KUKA KRL program: MyProgram_271().src

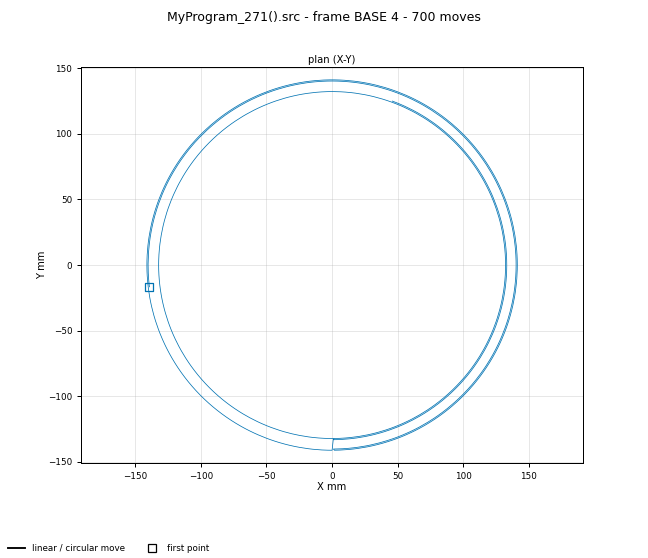
[picture p0: tool path of MyProgram_271().src in frame BASE 4, 700 of 700 moves have a stored position in this frame; points joined in program order, loops and branches not executed]
&ACCESS RVP
&REL 1
&PARAM TEMPLATE = C:\KRC\Roboter\Template\vorgabe
&PARAM EDITMASK = *
DEF MyProgram_271()
; ---- Setting reference (Base) ----
$BASE = BASE_DATA[4]

; --------------------------
; ---- Setting tool (TCP) ----
$TOOL = TOOL_DATA[3]
; --------------------------

$VEL.CP = VEL_APROX_PRINT
Startdeposition()
$VEL.CP = VEL_PRINT
LIN {X -139.2462,Y -16.5894,Z 170,A -172.5536,B 9.2163,C 0.2811,E1 9.0612,E2 264.1898} C_DIS
LIN {X -139.7898,Y -11.1357,Z 170,A -174.0658,B 9.2169,C 0.2622,E1 9.0608,E2 265.6084} C_DIS
LIN {X -140.1038,Y -5.997,Z 170,A -176.402,B 9.2169,C 0.2602,E1 9.0605,E2 267.9721} C_DIS
LIN {X -140.2304,Y 0.6703,Z 170,A -179.1601,B 9.2171,C 0.2528,E1 9.0604,E2 270.732} C_DIS
LIN {X -139.8512,Y 10.3146,Z 170,A 176.042,B 9.2171,C 0.2559,E1 9.0611,E2 275.6332} C_DIS
LIN {X -139.2175,Y 16.8301,Z 170,A 174.2066,B 9.2176,C 0.2339,E1 9.0617,E2 277.3608} C_DIS
LIN {X -138.6579,Y 20.951,Z 170,A 172.3266,B 9.2176,C 0.2321,E1 9.0624,E2 279.2619} C_DIS
LIN {X -137.8969,Y 25.4847,Z 170,A 170.0862,B 9.2176,C 0.2329,E1 9.0635,E2 281.5459} C_DIS
LIN {X -137.0475,Y 29.71,Z 170,A 168.7917,B 9.218,C 0.2199,E1 9.0643,E2 282.78} C_DIS
LIN {X -136.272,Y 33.0857,Z 170,A 167.3335,B 9.218,C 0.2166,E1 9.0652,E2 284.2422} C_DIS
LIN {X -135.2865,Y 36.9171,Z 170,A 165.7161,B 9.2181,C 0.2121,E1 9.0663,E2 285.8581} C_DIS
LIN {X -134.3405,Y 40.224,Z 170,A 164.2872,B 9.2182,C 0.2085,E1 9.0675,E2 287.2885} C_DIS
LIN {X -133.4935,Y 42.9443,Z 170,A 163.0667,B 9.2182,C 0.2062,E1 9.0685,E2 288.5149} C_DIS
LIN {X -132.1554,Y 46.9048,Z 170,A 161.2655,B 9.2183,C 0.2031,E1 9.0702,E2 290.3261} C_DIS
LIN {X -130.6875,Y 50.8469,Z 170,A 159.6638,B 9.2185,C 0.1964,E1 9.0717,E2 291.9111} C_DIS
LIN {X -129.48,Y 53.8478,Z 170,A 158.2691,B 9.2185,C 0.1941,E1 9.0732,E2 293.3137} C_DIS
LIN {X -128.0071,Y 57.2608,Z 170,A 156.6772,B 9.2185,C 0.1913,E1 9.075,E2 294.9132} C_DIS
LIN {X -126.4175,Y 60.6901,Z 170,A 155.1673,B 9.2187,C 0.1866,E1 9.0768,E2 296.4171} C_DIS
LIN {X -124.9093,Y 63.736,Z 170,A 153.7709,B 9.2187,C 0.1831,E1 9.0785,E2 297.813} C_DIS
LIN {X -123.2104,Y 66.9657,Z 170,A 152.1863,B 9.2187,C 0.1809,E1 9.0806,E2 299.4079} C_DIS
LIN {X -120.9477,Y 70.9706,Z 170,A 149.4715,B 9.2187,C 0.1905,E1 9.0846,E2 302.2246} C_DIS
LIN {X -117.5668,Y 76.4409,Z 170,A 147.5825,B 9.219,C 0.1713,E1 9.0873,E2 304.0192} C_DIS
LIN {X -114.9933,Y 80.2604,Z 170,A 145.6572,B 9.219,C 0.1675,E1 9.0904,E2 305.948} C_DIS
LIN {X -112.3015,Y 83.9859,Z 170,A 143.8132,B 9.2191,C 0.1624,E1 9.0934,E2 307.7859} C_DIS
LIN {X -109.5861,Y 87.4992,Z 170,A 142.121,B 9.2192,C 0.1561,E1 9.0963,E2 309.4609} C_DIS
LIN {X -107.3775,Y 90.1955,Z 170,A 140.1392,B 9.2192,C 0.1627,E1 9.0999,E2 311.5108} C_DIS
LIN {X -104.6541,Y 93.3422,Z 170,A 138.2237,B 9.2192,C 0.1627,E1 9.1036,E2 313.4514} C_DIS
LIN {X -101.1183,Y 97.1615,Z 170,A 136.7406,B 9.2194,C 0.1468,E1 9.1062,E2 314.8524} C_DIS
LIN {X -95.2851,Y 102.8885,Z 170,A 132.5478,B 9.2193,C 0.1552,E1 9.1149,E2 319.1478} C_DIS
LIN {X -90.8236,Y 106.8467,Z 170,A 130.8644,B 9.2195,C 0.137,E1 9.1183,E2 320.7354} C_DIS
LIN {X -85.4077,Y 111.2239,Z 170,A 127.4233,B 9.2195,C 0.1426,E1 9.126,E2 324.2479} C_DIS
LIN {X -81.5362,Y 114.0922,Z 170,A 126.3383,B 9.2197,C 0.1231,E1 9.1282,E2 325.221} C_DIS
LIN {X -77.667,Y 116.7607,Z 170,A 123.9376,B 9.2197,C 0.1287,E1 9.1338,E2 327.6801} C_DIS
LIN {X -74.607,Y 118.7394,Z 170,A 122.4708,B 9.2197,C 0.126,E1 9.1373,E2 329.1429} C_DIS
LIN {X -70.7584,Y 121.0724,Z 170,A 120.4134,B 9.2197,C 0.1272,E1 9.1423,E2 331.2259} C_DIS
LIN {X -67.873,Y 122.7128,Z 170,A 119.4128,B 9.2197,C 0.1187,E1 9.1446,E2 332.181} C_DIS
LIN {X -64.9436,Y 124.286,Z 170,A 117.9705,B 9.2198,C 0.1183,E1 9.1482,E2 333.6326} C_DIS
LIN {X -61.7916,Y 125.8828,Z 170,A 116.5014,B 9.2198,C 0.1169,E1 9.1519,E2 335.1037} C_DIS
LIN {X -56.515,Y 128.3407,Z 170,A 114.1253,B 9.2198,C 0.1139,E1 9.1579,E2 337.4776} C_DIS
LIN {X -53.1186,Y 129.7828,Z 170,A 112.3575,B 9.2198,C 0.1171,E1 9.1625,E2 339.2767} C_DIS
LIN {X -49.6846,Y 131.1348,Z 170,A 110.464,B 9.2198,C 0.1228,E1 9.1676,E2 341.2168} C_DIS
LIN {X -44.8258,Y 132.8743,Z 170,A 109.0846,B 9.2199,C 0.1069,E1 9.171,E2 342.5042} C_DIS
LIN {X -41.1545,Y 134.0558,Z 170,A 107.3834,B 9.2199,C 0.1079,E1 9.1756,E2 344.2198} C_DIS
LIN {X -37.5471,Y 135.1108,Z 170,A 105.8686,B 9.2199,C 0.1062,E1 9.1796,E2 345.731} C_DIS
LIN {X -34.4321,Y 135.9378,Z 170,A 104.5093,B 9.2199,C 0.106,E1 9.1833,E2 347.0947} C_DIS
LIN {X -30.7784,Y 136.8122,Z 170,A 102.9079,B 9.2199,C 0.1063,E1 9.1877,E2 348.7034} C_DIS
LIN {X -25.8795,Y 137.8229,Z 170,A 100.709,B 9.2199,C 0.1081,E1 9.1938,E2 350.9204} C_DIS
LIN {X -19.5101,Y 138.8675,Z 170,A 98.3717,B 9.22,C 0.101,E1 9.2001,E2 353.2186} C_DIS
LIN {X -16.5501,Y 139.2509,Z 170,A 97.0492,B 9.22,C 0.1025,E1 9.2038,E2 354.5533} C_DIS
LIN {X -12.8857,Y 139.6387,Z 170,A 95.4576,B 9.22,C 0.1038,E1 9.2083,E2 356.1548} C_DIS
LIN {X -8.0951,Y 139.9982,Z 170,A 93.4213,B 9.22,C 0.1048,E1 9.214,E2 358.1994} C_DIS
LIN {X -3.6352,Y 140.1842,Z 170,A 91.7596,B 9.22,C 0.1013,E1 9.2185,E2 359.8399} C_DIS
LIN {X 0.3041,Y 140.2316,Z 170,A 90.0873,B 9.22,C 0.1025,E1 9.2232,E2 361.5193} C_DIS
LIN {X 4.399,Y 140.163,Z 170,A 88.3947,B 9.22,C 0.103,E1 9.228,E2 363.2136} C_DIS
LIN {X 8.9248,Y 139.9471,Z 170,A 86.62,B 9.22,C 0.1017,E1 9.2329,E2 364.9779} C_DIS
LIN {X 12.8173,Y 139.6452,Z 170,A 84.9722,B 9.22,C 0.1031,E1 9.2375,E2 366.6318} C_DIS
LIN {X 17.1727,Y 139.1766,Z 170,A 83.2612,B 9.22,C 0.1021,E1 9.2422,E2 368.3323} C_DIS
LIN {X 20.6785,Y 138.7001,Z 170,A 81.5426,B 9.22,C 0.1082,E1 9.247,E2 370.0846} C_DIS
LIN {X 24.8793,Y 138.0063,Z 170,A 80.0499,B 9.22,C 0.1039,E1 9.2511,E2 371.5459} C_DIS
LIN {X 28.565,Y 137.292,Z 170,A 78.4857,B 9.22,C 0.1054,E1 9.2553,E2 373.1135} C_DIS
LIN {X 35.6917,Y 135.6133,Z 170,A 75.7106,B 9.22,C 0.1029,E1 9.2628,E2 375.8608} C_DIS
LIN {X 39.6337,Y 134.5135,Z 170,A 73.9278,B 9.22,C 0.1065,E1 9.2676,E2 377.6572} C_DIS
LIN {X 42.5414,Y 133.6222,Z 170,A 72.6579,B 9.22,C 0.1081,E1 9.271,E2 378.9303} C_DIS
LIN {X 46.1819,Y 132.4082,Z 170,A 71.0986,B 9.22,C 0.1093,E1 9.2751,E2 380.4884} C_DIS
LIN {X 49.4224,Y 131.233,Z 170,A 69.6904,B 9.2199,C 0.1107,E1 9.2788,E2 381.8964} C_DIS
LIN {X 53.2544,Y 129.7278,Z 170,A 67.7835,B 9.2199,C 0.1173,E1 9.2839,E2 383.8314} C_DIS
LIN {X 57.511,Y 127.8952,Z 170,A 66.1229,B 9.2199,C 0.1145,E1 9.288,E2 385.4627} C_DIS
LIN {X 61.3313,Y 126.1098,Z 170,A 63.7761,B 9.2196,C 0.13,E1 9.2941,E2 387.8874} C_DIS
LIN {X 66.1302,Y 123.661,Z 170,A 62.381,B 9.2198,C 0.1155,E1 9.2973,E2 389.1818} C_DIS
LIN {X 68.9326,Y 122.1209,Z 170,A 60.8762,B 9.2198,C 0.1216,E1 9.3011,E2 390.7116} C_DIS
LIN {X 72.6923,Y 119.9209,Z 170,A 59.0261,B 9.2198,C 0.1258,E1 9.3055,E2 392.5707} C_DIS
LIN {X 75.8926,Y 117.922,Z 170,A 57.5682,B 9.2197,C 0.1263,E1 9.3089,E2 394.0183} C_DIS
LIN {X 83.3663,Y 112.7626,Z 170,A 54.1374,B 9.2197,C 0.1263,E1 9.3167,E2 397.4145} C_DIS
LIN {X 87.4079,Y 109.6587,Z 170,A 51.83,B 9.2196,C 0.1349,E1 9.3219,E2 399.7509} C_DIS
LIN {X 90.8036,Y 106.8638,Z 170,A 50.0554,B 9.2196,C 0.1377,E1 9.3257,E2 401.5231} C_DIS
LIN {X 94.272,Y 103.8169,Z 170,A 48.2485,B 9.2196,C 0.1395,E1 9.3294,E2 403.3205} C_DIS
LIN {X 97.1834,Y 101.0976,Z 170,A 46.6007,B 9.2195,C 0.1432,E1 9.3327,E2 404.9714} C_DIS
LIN {X 100.2842,Y 98.0219,Z 170,A 44.8365,B 9.2195,C 0.1463,E1 9.3362,E2 406.7336} C_DIS
LIN {X 103.2198,Y 94.9254,Z 170,A 43.0036,B 9.2193,C 0.152,E1 9.3397,E2 408.5784} C_DIS
LIN {X 106.1594,Y 91.6262,Z 170,A 41.2904,B 9.2193,C 0.1538,E1 9.3429,E2 410.2808} C_DIS
LIN {X 109.1335,Y 88.0626,Z 170,A 39.4373,B 9.2193,C 0.157,E1 9.3461,E2 412.1291} C_DIS
LIN {X 111.9131,Y 84.5022,Z 170,A 37.6022,B 9.2192,C 0.161,E1 9.3493,E2 413.9637} C_DIS
LIN {X 114.6849,Y 80.7004,Z 170,A 35.7168,B 9.2191,C 0.1647,E1 9.3523,E2 415.8454} C_DIS
LIN {X 117.5997,Y 76.3903,Z 170,A 33.8456,B 9.2191,C 0.1639,E1 9.3552,E2 417.6854} C_DIS
LIN {X 121.414,Y 70.17,Z 170,A 30.7692,B 9.2189,C 0.1735,E1 9.3597,E2 420.7758} C_DIS
LIN {X 123.347,Y 66.7145,Z 170,A 29.0536,B 9.2189,C 0.1798,E1 9.362,E2 422.5048} C_DIS
LIN {X 125.1484,Y 63.2663,Z 170,A 27.5598,B 9.2188,C 0.1816,E1 9.3639,E2 423.9873} C_DIS
LIN {X 127.464,Y 58.4612,Z 170,A 25.3654,B 9.2187,C 0.1877,E1 9.3665,E2 426.1851} C_DIS
LIN {X 130.2216,Y 52.0303,Z 170,A 22.604,B 9.2186,C 0.193,E1 9.3695,E2 428.9361} C_DIS
LIN {X 131.5973,Y 48.4498,Z 170,A 21.1227,B 9.2186,C 0.1952,E1 9.3709,E2 430.4076} C_DIS
LIN {X 133.1157,Y 44.101,Z 170,A 19.2332,B 9.2184,C 0.2005,E1 9.3727,E2 432.2994} C_DIS
LIN {X 134.2,Y 40.6834,Z 170,A 17.8197,B 9.2184,C 0.2034,E1 9.3738,E2 433.7075} C_DIS
LIN {X 135.0818,Y 37.6509,Z 170,A 16.5285,B 9.2182,C 0.207,E1 9.3748,E2 434.9998} C_DIS
LIN {X 135.9488,Y 34.3891,Z 170,A 15.162,B 9.2182,C 0.2105,E1 9.3758,E2 436.3657} C_DIS
LIN {X 137.2404,Y 28.8166,Z 170,A 12.8741,B 9.218,C 0.216,E1 9.3772,E2 438.6494} C_DIS
LIN {X 137.8314,Y 25.8349,Z 170,A 11.6299,B 9.218,C 0.2196,E1 9.3778,E2 439.8948} C_DIS
LIN {X 138.8688,Y 19.5011,Z 170,A 8.9512,B 9.2177,C 0.2284,E1 9.379,E2 442.583} C_DIS
LIN {X 139.473,Y 14.5673,Z 170,A 7.1046,B 9.2177,C 0.2299,E1 9.3796,E2 444.4078} C_DIS
LIN {X 139.77,Y 11.3697,Z 170,A 5.7499,B 9.2176,C 0.2347,E1 9.3799,E2 445.7692} C_DIS
LIN {X 140.0376,Y 7.3716,Z 170,A 4.0974,B 9.2175,C 0.2398,E1 9.3802,E2 447.4251} C_DIS
LIN {X 140.1978,Y 3.1337,Z 170,A 2.476,B 9.2174,C 0.2422,E1 9.3803,E2 449.0338} C_DIS
LIN {X 140.2322,Y -0.3501,Z 170,A 0.9312,B 9.2172,C 0.2492,E1 9.3803,E2 450.5955} C_DIS
LIN {X 140.161,Y -4.4688,Z 170,A -0.6532,B 9.2172,C 0.2518,E1 9.3803,E2 452.1689} C_DIS
LIN {X 139.9543,Y -8.8077,Z 170,A -2.3812,B 9.217,C 0.2558,E1 9.38,E2 453.8925} C_DIS
LIN {X 139.5984,Y -13.3047,Z 170,A -4.1955,B 9.217,C 0.2605,E1 9.3796,E2 455.7049} C_DIS
LIN {X 139.192,Y -17.0436,Z 170,A -5.6897,B 9.2168,C 0.264,E1 9.3791,E2 457.1953} C_DIS
LIN {X 138.6832,Y -20.7877,Z 170,A -7.2663,B 9.2167,C 0.2692,E1 9.3785,E2 458.7776} C_DIS
LIN {X 138.0405,Y -24.6885,Z 170,A -8.7749,B 9.2166,C 0.2713,E1 9.3777,E2 460.274} C_DIS
LIN {X 137.1856,Y -29.0702,Z 170,A -10.4751,B 9.2166,C 0.2736,E1 9.3768,E2 461.9602} C_DIS
LIN {X 135.6171,Y -35.6776,Z 170,A -13.2274,B 9.2163,C 0.281,E1 9.375,E2 464.7124} C_DIS
LIN {X 134.0219,Y -41.2653,Z 170,A -15.6706,B 9.2161,C 0.2893,E1 9.3731,E2 467.1671} C_DIS
LIN {X 132.9867,Y -44.4884,Z 170,A -17.0306,B 9.2159,C 0.2926,E1 9.3719,E2 468.5255} C_DIS
LIN {X 131.8302,Y -47.8069,Z 170,A -18.5104,B 9.2158,C 0.2977,E1 9.3705,E2 470.0125} C_DIS
LIN {X 130.5867,Y -51.1062,Z 170,A -19.8379,B 9.2158,C 0.299,E1 9.3692,E2 471.3269} C_DIS
LIN {X 129.3454,Y -54.1702,Z 170,A -21.2108,B 9.2156,C 0.3032,E1 9.3678,E2 472.7041} C_DIS
LIN {X 127.9157,Y -57.465,Z 170,A -22.9582,B 9.2153,C 0.3137,E1 9.3657,E2 474.4893} C_DIS
LIN {X 126.4198,Y -60.6854,Z 170,A -24.0769,B 9.2153,C 0.3098,E1 9.3644,E2 475.5666} C_DIS
LIN {X 124.715,Y -64.1177,Z 170,A -25.7281,B 9.2152,C 0.3159,E1 9.3623,E2 477.2305} C_DIS
LIN {X 122.4608,Y -68.328,Z 170,A -27.6302,B 9.2151,C 0.3198,E1 9.3598,E2 479.1284} C_DIS
LIN {X 120.1993,Y -72.2318,Z 170,A -29.4704,B 9.2149,C 0.3245,E1 9.3572,E2 480.97} C_DIS
LIN {X 117.3839,Y -76.7225,Z 170,A -31.3303,B 9.2149,C 0.3227,E1 9.3545,E2 482.7925} C_DIS
LIN {X 115.7561,Y -79.1564,Z 170,A -33.1166,B 9.2144,C 0.3395,E1 9.3515,E2 484.6566} C_DIS
LIN {X 113.2796,Y -82.6625,Z 170,A -34.6544,B 9.2144,C 0.3387,E1 9.349,E2 486.1683} C_DIS
LIN {X 109.4132,Y -87.7159,Z 170,A -37.0166,B 9.2144,C 0.3393,E1 9.345,E2 488.5024} C_DIS
LIN {X 106.6746,Y -91.0262,Z 170,A -38.7536,B 9.2142,C 0.3429,E1 9.3419,E2 490.2388} C_DIS
LIN {X 103.7265,Y -94.3716,Z 170,A -40.6773,B 9.214,C 0.3493,E1 9.3383,E2 492.1776} C_DIS
LIN {X 100.1033,Y -98.2064,Z 170,A -42.7047,B 9.214,C 0.3511,E1 9.3344,E2 494.1905} C_DIS
LIN {X 96.9043,Y -101.3643,Z 170,A -44.5337,B 9.2138,C 0.3548,E1 9.3308,E2 496.0204} C_DIS
LIN {X 93.6356,Y -104.3913,Z 170,A -46.3608,B 9.2136,C 0.3586,E1 9.327,E2 497.8502} C_DIS
LIN {X 90.3082,Y -107.283,Z 170,A -47.8776,B 9.2137,C 0.3557,E1 9.3238,E2 499.3316} C_DIS
LIN {X 88.0101,Y -109.1759,Z 170,A -49.3011,B 9.2135,C 0.3628,E1 9.3207,E2 500.7834} C_DIS
LIN {X 84.3759,Y -112.0084,Z 170,A -51.1773,B 9.2133,C 0.3661,E1 9.3165,E2 502.6605} C_DIS
LIN {X 80.817,Y -114.6027,Z 170,A -53.2245,B 9.213,C 0.3749,E1 9.3118,E2 504.7416} C_DIS
LIN {X 77.7606,Y -116.6982,Z 170,A -54.0819,B 9.2135,C 0.3627,E1 9.31,E2 505.5149} C_DIS
LIN {X 72.9752,Y -119.7495,Z 170,A -57.1785,B 9.2126,C 0.384,E1 9.3024,E2 508.7149} C_DIS
LIN {X 69.0385,Y -122.0614,Z 170,A -58.3441,B 9.2131,C 0.3712,E1 9.2999,E2 509.7911} C_DIS
LIN {X 66.5378,Y -123.442,Z 170,A -59.7489,B 9.2129,C 0.3783,E1 9.2963,E2 511.228} C_DIS
LIN {X 62.943,Y -125.313,Z 170,A -61.53,B 9.2126,C 0.3835,E1 9.2918,E2 513.0269} C_DIS
LIN {X 59.5131,Y -126.9776,Z 170,A -63.5999,B 9.2121,C 0.3969,E1 9.2865,E2 515.1644} C_DIS
LIN {X 54.2623,Y -129.3069,Z 170,A -64.9711,B 9.2129,C 0.3783,E1 9.2832,E2 516.4107} C_DIS
LIN {X 50.1462,Y -130.9599,Z 170,A -66.9993,B 9.2126,C 0.3852,E1 9.2779,E2 518.4687} C_DIS
LIN {X 47.0424,Y -132.1058,Z 170,A -68.3547,B 9.2126,C 0.3868,E1 9.2743,E2 519.8256} C_DIS
LIN {X 42.2849,Y -133.7041,Z 170,A -70.3597,B 9.2125,C 0.3879,E1 9.269,E2 521.8263} C_DIS
LIN {X 39.1077,Y -134.6675,Z 170,A -71.7116,B 9.2125,C 0.3891,E1 9.2654,E2 523.1785} C_DIS
LIN {X 35.9768,Y -135.5373,Z 170,A -73.3749,B 9.2121,C 0.3975,E1 9.2608,E2 524.8864} C_DIS
LIN {X 32.5199,Y -136.4084,Z 170,A -74.4884,B 9.2123,C 0.3913,E1 9.2579,E2 525.9563} C_DIS
LIN {X 29.3843,Y -137.1178,Z 170,A -75.8357,B 9.2123,C 0.393,E1 9.2542,E2 527.3089} C_DIS
LIN {X 25.6891,Y -137.8593,Z 170,A -77.4109,B 9.2122,C 0.3948,E1 9.2499,E2 528.8897} C_DIS
LIN {X 19.4617,Y -138.8744,Z 170,A -79.9112,B 9.2122,C 0.3946,E1 9.243,E2 531.3815} C_DIS
LIN {X 16.2153,Y -139.2909,Z 170,A -81.2556,B 9.2122,C 0.3954,E1 9.2393,E2 532.7275} C_DIS
LIN {X 12.2333,Y -139.6971,Z 170,A -82.962,B 9.2121,C 0.3976,E1 9.2345,E2 534.4442} C_DIS
LIN {X 7.9939,Y -140.0044,Z 170,A -84.7136,B 9.2121,C 0.3984,E1 9.2296,E2 536.1986} C_DIS
LIN {X 3.7131,Y -140.182,Z 170,A -86.3843,B 9.2121,C 0.3971,E1 9.225,E2 537.8598} C_DIS
LIN {X 1.0099,Y -140.2255,Z 170,A -87.3545,B 9.2121,C 0.3945,E1 9.2223,E2 538.8129} C_DIS
Enddeposition()
LIN {X 1.0099,Y -140.2255,Z 170,A -87.3545,B 9.2121,C 0.3945,E1 9.2223,E2 538.8129} C_DIS
Startdeposition()
$VEL.CP = VEL_PRINT
LIN {X 1.7317,Y -141.1336,Z 170,A -86.5013,B 9.2127,C 0.388,E1 9.225,E2 537.9198} C_DIS
LIN {X 6.0081,Y -141.0158,Z 170,A -84.7676,B 9.2127,C 0.3877,E1 9.2298,E2 536.1856} C_DIS
LIN {X 9.5773,Y -140.8192,Z 170,A -83.3221,B 9.2127,C 0.3874,E1 9.2339,E2 534.7401} C_DIS
LIN {X 12.9203,Y -140.5513,Z 170,A -81.9666,B 9.2127,C 0.387,E1 9.2376,E2 533.3846} C_DIS
LIN {X 16.3651,Y -140.1912,Z 170,A -80.5449,B 9.2127,C 0.386,E1 9.2416,E2 531.96} C_DIS
LIN {X 19.9142,Y -139.7308,Z 170,A -79.1269,B 9.2127,C 0.386,E1 9.2455,E2 530.5458} C_DIS
LIN {X 23.335,Y -139.2003,Z 170,A -77.7449,B 9.2127,C 0.3857,E1 9.2493,E2 529.1659} C_DIS
LIN {X 26.7407,Y -138.5866,Z 170,A -76.3301,B 9.2128,C 0.3846,E1 9.2532,E2 527.7489} C_DIS
LIN {X 30.1968,Y -137.8751,Z 170,A -74.7717,B 9.213,C 0.3808,E1 9.2575,E2 526.1729} C_DIS
LIN {X 34.285,Y -136.9159,Z 170,A -73.1966,B 9.213,C 0.3822,E1 9.2617,E2 524.6138} C_DIS
LIN {X 38.4284,Y -135.8111,Z 170,A -71.4722,B 9.213,C 0.3811,E1 9.2664,E2 522.8903} C_DIS
LIN {X 42.4547,Y -134.607,Z 170,A -69.724,B 9.213,C 0.3785,E1 9.2711,E2 521.1353} C_DIS
LIN {X 45.925,Y -133.4623,Z 170,A -68.2993,B 9.213,C 0.3782,E1 9.2748,E2 519.7172} C_DIS
LIN {X 49.1829,Y -132.2964,Z 170,A -66.904,B 9.2131,C 0.3769,E1 9.2785,E2 518.3222} C_DIS
LIN {X 52.4108,Y -131.0512,Z 170,A -65.4233,B 9.2133,C 0.3735,E1 9.2824,E2 516.8301} C_DIS
LIN {X 56.3656,Y -129.3995,Z 170,A -63.7356,B 9.2133,C 0.3725,E1 9.2867,E2 515.148} C_DIS
LIN {X 60.3477,Y -127.5916,Z 170,A -62.0128,B 9.2133,C 0.3713,E1 9.291,E2 513.4308} C_DIS
LIN {X 63.4608,Y -126.0725,Z 170,A -60.5217,B 9.2135,C 0.3674,E1 9.2948,E2 511.9271} C_DIS
LIN {X 66.9422,Y -124.2598,Z 170,A -58.9748,B 9.2135,C 0.3662,E1 9.2986,E2 510.3851} C_DIS
LIN {X 70.688,Y -122.1676,Z 170,A -57.2428,B 9.2136,C 0.3637,E1 9.3028,E2 508.6528} C_DIS
LIN {X 74.4416,Y -119.9174,Z 170,A -55.4816,B 9.2137,C 0.3612,E1 9.307,E2 506.8921} C_DIS
LIN {X 78.0338,Y -117.6121,Z 170,A -53.7397,B 9.2139,C 0.3581,E1 9.3111,E2 505.1473} C_DIS
LIN {X 81.6517,Y -115.1297,Z 170,A -51.9924,B 9.2139,C 0.3557,E1 9.3151,E2 503.4029} C_DIS
LIN {X 85.1033,Y -112.6017,Z 170,A -50.2862,B 9.2141,C 0.3532,E1 9.3189,E2 501.6991} C_DIS
LIN {X 88.5132,Y -109.9415,Z 170,A -48.5373,B 9.2141,C 0.3501,E1 9.3227,E2 499.9494} C_DIS
LIN {X 91.8473,Y -107.1723,Z 170,A -46.7828,B 9.2143,C 0.3467,E1 9.3265,E2 498.1938} C_DIS
LIN {X 95.0903,Y -104.3056,Z 170,A -45.0499,B 9.2144,C 0.3437,E1 9.3301,E2 496.4624} C_DIS
LIN {X 98.3293,Y -101.2576,Z 170,A -43.3047,B 9.2144,C 0.3414,E1 9.3336,E2 494.7234} C_DIS
LIN {X 101.3041,Y -98.2812,Z 170,A -41.5824,B 9.2146,C 0.3374,E1 9.337,E2 492.9975} C_DIS
LIN {X 104.3111,Y -95.0842,Z 170,A -39.8215,B 9.2148,C 0.3339,E1 9.3403,E2 491.2377} C_DIS
LIN {X 107.1771,Y -91.8418,Z 170,A -38.0904,B 9.2148,C 0.3305,E1 9.3435,E2 489.5081} C_DIS
LIN {X 109.9417,Y -88.5129,Z 170,A -36.3712,B 9.215,C 0.3274,E1 9.3465,E2 487.7921} C_DIS
LIN {X 112.6208,Y -85.078,Z 170,A -34.6202,B 9.2151,C 0.3236,E1 9.3495,E2 486.0415} C_DIS
LIN {X 115.1411,Y -81.6355,Z 170,A -32.888,B 9.2153,C 0.3194,E1 9.3523,E2 484.3074} C_DIS
LIN {X 117.6126,Y -78.033,Z 170,A -31.1053,B 9.2154,C 0.3148,E1 9.3551,E2 482.5217} C_DIS
LIN {X 120.165,Y -74.0417,Z 170,A -29.2455,B 9.2155,C 0.3115,E1 9.3578,E2 480.6683} C_DIS
LIN {X 122.3787,Y -70.3232,Z 170,A -27.5023,B 9.2157,C 0.3073,E1 9.3603,E2 478.925} C_DIS
LIN {X 124.4786,Y -66.5348,Z 170,A -25.7885,B 9.2158,C 0.3038,E1 9.3626,E2 477.2153} C_DIS
LIN {X 126.4581,Y -62.6863,Z 170,A -24.1374,B 9.2158,C 0.3017,E1 9.3646,E2 475.5762} C_DIS
LIN {X 127.9637,Y -59.553,Z 170,A -22.7472,B 9.216,C 0.2984,E1 9.3663,E2 474.1872} C_DIS
LIN {X 129.4045,Y -56.3541,Z 170,A -21.2293,B 9.2162,C 0.2923,E1 9.368,E2 472.6555} C_DIS
LIN {X 131.0906,Y -52.313,Z 170,A -19.4702,B 9.2163,C 0.2879,E1 9.3699,E2 470.897} C_DIS
LIN {X 132.5808,Y -48.4132,Z 170,A -17.9207,B 9.2163,C 0.2867,E1 9.3714,E2 469.3648} C_DIS
LIN {X 133.7623,Y -45.045,Z 170,A -16.5228,B 9.2164,C 0.2839,E1 9.3726,E2 467.9721} C_DIS
LIN {X 134.8313,Y -41.7363,Z 170,A -15.1015,B 9.2166,C 0.2797,E1 9.3738,E2 466.5481} C_DIS
LIN {X 135.8147,Y -38.4155,Z 170,A -13.7164,B 9.2166,C 0.2763,E1 9.3749,E2 465.1642} C_DIS
LIN {X 136.7157,Y -35.0736,Z 170,A -12.2217,B 9.2168,C 0.2701,E1 9.376,E2 463.6563} C_DIS
LIN {X 137.7149,Y -30.921,Z 170,A -10.6326,B 9.2168,C 0.2687,E1 9.377,E2 462.0845} C_DIS
LIN {X 138.4337,Y -27.5269,Z 170,A -9.2493,B 9.217,C 0.2652,E1 9.3777,E2 460.703} C_DIS
LIN {X 139.0676,Y -24.1251,Z 170,A -7.8686,B 9.217,C 0.2618,E1 9.3784,E2 459.3241} C_DIS
LIN {X 139.6174,Y -20.7074,Z 170,A -6.4624,B 9.2172,C 0.2577,E1 9.379,E2 457.9164} C_DIS
LIN {X 140.0824,Y -17.2771,Z 170,A -5.0817,B 9.2172,C 0.2542,E1 9.3795,E2 456.5375} C_DIS
LIN {X 140.4632,Y -13.838,Z 170,A -3.7012,B 9.2174,C 0.2507,E1 9.3799,E2 455.1587} C_DIS
LIN {X 140.7605,Y -10.3822,Z 170,A -2.3229,B 9.2174,C 0.2473,E1 9.3802,E2 453.7829} C_DIS
LIN {X 140.9732,Y -6.9206,Z 170,A -0.9451,B 9.2176,C 0.244,E1 9.3804,E2 452.4077} C_DIS
LIN {X 141.1011,Y -3.4627,Z 170,A 0.427,B 9.2176,C 0.2407,E1 9.3805,E2 451.0385} C_DIS
LIN {X 141.1449,Y 0.1953,Z 170,A 1.8961,B 9.2178,C 0.2367,E1 9.3805,E2 449.5702} C_DIS
LIN {X 141.0784,Y 4.2791,Z 170,A 3.5618,B 9.2178,C 0.2317,E1 9.3805,E2 447.9019} C_DIS
LIN {X 140.9197,Y 7.9655,Z 170,A 5.1114,B 9.218,C 0.2261,E1 9.3802,E2 446.3442} C_DIS
LIN {X 140.691,Y 11.2994,Z 170,A 6.3317,B 9.218,C 0.2255,E1 9.38,E2 445.1405} C_DIS
LIN {X 140.3569,Y 14.8749,Z 170,A 7.8855,B 9.2182,C 0.219,E1 9.3795,E2 443.5727} C_DIS
LIN {X 139.7992,Y 19.4351,Z 170,A 9.503,B 9.2182,C 0.2196,E1 9.379,E2 441.9861} C_DIS
LIN {X 139.3517,Y 22.4275,Z 170,A 10.8391,B 9.2183,C 0.2135,E1 9.3784,E2 440.6348} C_DIS
LIN {X 138.7596,Y 25.8356,Z 170,A 12.2181,B 9.2183,C 0.2101,E1 9.3777,E2 439.2579} C_DIS
LIN {X 138.0849,Y 29.2252,Z 170,A 13.5968,B 9.2185,C 0.2066,E1 9.3769,E2 437.8812} C_DIS
LIN {X 137.2051,Y 33.1057,Z 170,A 15.2249,B 9.2185,C 0.2018,E1 9.3759,E2 436.25} C_DIS
LIN {X 136.2727,Y 36.7577,Z 170,A 16.7514,B 9.2187,C 0.1976,E1 9.3748,E2 434.7228} C_DIS
LIN {X 135.0645,Y 40.9743,Z 170,A 18.4444,B 9.2187,C 0.1947,E1 9.3735,E2 433.0399} C_DIS
LIN {X 134.0187,Y 44.275,Z 170,A 19.8278,B 9.2187,C 0.1914,E1 9.3723,E2 431.6583} C_DIS
LIN {X 132.8926,Y 47.5485,Z 170,A 21.2132,B 9.2189,C 0.1881,E1 9.371,E2 430.2744} C_DIS
LIN {X 131.6847,Y 50.798,Z 170,A 22.6024,B 9.2189,C 0.1847,E1 9.3696,E2 428.8865} C_DIS
LIN {X 130.3935,Y 54.0264,Z 170,A 23.9868,B 9.2189,C 0.1816,E1 9.3682,E2 427.5047} C_DIS
LIN {X 129.0328,Y 57.2006,Z 170,A 25.3751,B 9.2191,C 0.1782,E1 9.3666,E2 426.1172} C_DIS
LIN {X 127.5948,Y 60.341,Z 170,A 26.7514,B 9.2191,C 0.1751,E1 9.365,E2 424.7433} C_DIS
LIN {X 126.0726,Y 63.4606,Z 170,A 28.2427,B 9.2192,C 0.1695,E1 9.3632,E2 423.2404} C_DIS
LIN {X 124.0681,Y 67.2973,Z 170,A 29.9578,B 9.2192,C 0.1661,E1 9.3609,E2 421.5298} C_DIS
LIN {X 121.9391,Y 71.0827,Z 170,A 31.7004,B 9.2193,C 0.1622,E1 9.3585,E2 419.7888} C_DIS
LIN {X 119.7044,Y 74.7838,Z 170,A 33.4266,B 9.2194,C 0.1585,E1 9.356,E2 418.0654} C_DIS
LIN {X 117.3558,Y 78.4177,Z 170,A 35.1402,B 9.2194,C 0.1553,E1 9.3533,E2 416.3564} C_DIS
LIN {X 114.8961,Y 81.9794,Z 170,A 36.8861,B 9.2195,C 0.1514,E1 9.3505,E2 414.6111} C_DIS
LIN {X 112.3285,Y 85.4643,Z 170,A 38.6419,B 9.2195,C 0.1474,E1 9.3476,E2 412.8546} C_DIS
LIN {X 109.6548,Y 88.8687,Z 170,A 40.3617,B 9.2196,C 0.1444,E1 9.3446,E2 411.1388} C_DIS
LIN {X 106.878,Y 92.189,Z 170,A 42.0907,B 9.2196,C 0.1412,E1 9.3415,E2 409.4127} C_DIS
LIN {X 103.9933,Y 95.4312,Z 170,A 43.8407,B 9.2197,C 0.1377,E1 9.3382,E2 407.6635} C_DIS
LIN {X 101.0203,Y 98.5735,Z 170,A 45.5915,B 9.2197,C 0.1342,E1 9.3348,E2 405.9128} C_DIS
LIN {X 97.9517,Y 101.6232,Z 170,A 47.3099,B 9.2198,C 0.1315,E1 9.3314,E2 404.1987} C_DIS
LIN {X 94.7913,Y 104.5769,Z 170,A 49.0407,B 9.2198,C 0.1287,E1 9.3278,E2 402.4706} C_DIS
LIN {X 91.5315,Y 107.4417,Z 170,A 50.7972,B 9.2199,C 0.1255,E1 9.3241,E2 400.7143} C_DIS
LIN {X 88.1943,Y 110.1981,Z 170,A 52.5412,B 9.2199,C 0.1226,E1 9.3204,E2 398.9716} C_DIS
LIN {X 84.7733,Y 112.8507,Z 170,A 54.286,B 9.2199,C 0.1199,E1 9.3165,E2 397.228} C_DIS
LIN {X 81.261,Y 115.4053,Z 170,A 56.012,B 9.22,C 0.1178,E1 9.3126,E2 395.5065} C_DIS
LIN {X 77.5358,Y 117.9403,Z 170,A 57.7927,B 9.22,C 0.1159,E1 9.3085,E2 393.7318} C_DIS
LIN {X 74.0413,Y 120.1652,Z 170,A 59.5129,B 9.22,C 0.1125,E1 9.3044,E2 392.0064} C_DIS
LIN {X 70.3224,Y 122.3792,Z 170,A 61.2669,B 9.2201,C 0.1101,E1 9.3001,E2 390.2528} C_DIS
LIN {X 66.5235,Y 124.4847,Z 170,A 63.0104,B 9.2201,C 0.1081,E1 9.2959,E2 388.5116} C_DIS
LIN {X 62.6699,Y 126.4662,Z 170,A 64.6617,B 9.2201,C 0.1082,E1 9.2918,E2 386.874} C_DIS
LIN {X 59.5559,Y 127.9624,Z 170,A 66.0545,B 9.2201,C 0.1067,E1 9.2883,E2 385.4825} C_DIS
LIN {X 56.3566,Y 129.4033,Z 170,A 67.4427,B 9.2201,C 0.1059,E1 9.2847,E2 384.0991} C_DIS
LIN {X 53.1624,Y 130.7483,Z 170,A 68.8706,B 9.2201,C 0.1039,E1 9.2811,E2 382.6685} C_DIS
LIN {X 50.0365,Y 131.9767,Z 170,A 70.2271,B 9.2201,C 0.1027,E1 9.2775,E2 381.3131} C_DIS
LIN {X 46.7831,Y 133.1648,Z 170,A 71.6568,B 9.2202,C 0.1008,E1 9.2738,E2 379.8805} C_DIS
LIN {X 43.5013,Y 134.2727,Z 170,A 73.0566,B 9.2202,C 0.0997,E1 9.27,E2 378.4816} C_DIS
LIN {X 40.0923,Y 135.3293,Z 170,A 74.4708,B 9.2202,C 0.0993,E1 9.2663,E2 377.0721} C_DIS
LIN {X 36.7501,Y 136.2747,Z 170,A 75.8751,B 9.2202,C 0.0983,E1 9.2625,E2 375.6688} C_DIS
LIN {X 33.4994,Y 137.1102,Z 170,A 77.2335,B 9.2202,C 0.0975,E1 9.2588,E2 374.3113} C_DIS
LIN {X 30.1256,Y 137.8905,Z 170,A 78.6343,B 9.2202,C 0.0967,E1 9.255,E2 372.9114} C_DIS
LIN {X 26.7351,Y 138.5876,Z 170,A 80.0557,B 9.2202,C 0.0956,E1 9.2511,E2 371.4883} C_DIS
LIN {X 23.3246,Y 139.2021,Z 170,A 81.4358,B 9.2202,C 0.0956,E1 9.2473,E2 370.1119} C_DIS
LIN {X 19.9035,Y 139.7323,Z 170,A 82.8352,B 9.2202,C 0.0951,E1 9.2435,E2 368.7138} C_DIS
LIN {X 16.3629,Y 140.1915,Z 170,A 84.2752,B 9.2202,C 0.0948,E1 9.2395,E2 367.2755} C_DIS
LIN {X 12.6498,Y 140.5769,Z 170,A 85.7877,B 9.2202,C 0.0945,E1 9.2353,E2 365.764} C_DIS
LIN {X 9.3852,Y 140.8322,Z 170,A 87.1188,B 9.2202,C 0.0942,E1 9.2316,E2 364.4331} C_DIS
LIN {X 6.0058,Y 141.0159,Z 170,A 88.6485,B 9.2203,C 0.0908,E1 9.2272,E2 362.884} C_DIS
LIN {X 1.7276,Y 141.1337,Z 170,A 90.3187,B 9.2203,C 0.0922,E1 9.2226,E2 361.2232} C_DIS
LIN {X -1.734,Y 141.1336,Z 170,A 91.8057,B 9.2203,C 0.0906,E1 9.2184,E2 359.7264} C_DIS
LIN {X -6.3426,Y 141.0022,Z 170,A 93.5006,B 9.2203,C 0.0944,E1 9.2138,E2 358.055} C_DIS
LIN {X -9.5773,Y 140.8192,Z 170,A 94.8469,B 9.2203,C 0.094,E1 9.21,E2 356.7054} C_DIS
LIN {X -12.9211,Y 140.5512,Z 170,A 96.3436,B 9.2203,C 0.0917,E1 9.2058,E2 355.1921} C_DIS
LIN {X -17.2795,Y 140.0821,Z 170,A 97.966,B 9.2203,C 0.0955,E1 9.2013,E2 353.5909} C_DIS
LIN {X -20.7608,Y 139.6098,Z 170,A 99.4201,B 9.2203,C 0.0955,E1 9.1973,E2 352.134} C_DIS
LIN {X -24.226,Y 139.0495,Z 170,A 100.8573,B 9.2203,C 0.096,E1 9.1934,E2 350.6962} C_DIS
LIN {X -27.732,Y 138.392,Z 170,A 102.4356,B 9.2203,C 0.0943,E1 9.189,E2 349.1021} C_DIS
LIN {X -32.6185,Y 137.3225,Z 170,A 104.3313,B 9.2203,C 0.0983,E1 9.1839,E2 347.2249} C_DIS
LIN {X -36.7599,Y 136.2721,Z 170,A 106.0676,B 9.2203,C 0.0996,E1 9.1792,E2 345.4895} C_DIS
LIN {X -40.0924,Y 135.3292,Z 170,A 107.5106,B 9.2203,C 0.1,E1 9.1753,E2 344.0428} C_DIS
LIN {X -44.274,Y 134.0191,Z 170,A 109.2773,B 9.2203,C 0.1019,E1 9.1706,E2 342.2789} C_DIS
LIN {X -47.5753,Y 132.8829,Z 170,A 110.6938,B 9.2202,C 0.1033,E1 9.1669,E2 340.8636} C_DIS
LIN {X -50.8146,Y 131.6783,Z 170,A 112.1037,B 9.2202,C 0.1047,E1 9.1632,E2 339.4539} C_DIS
LIN {X -54.0207,Y 130.3959,Z 170,A 113.5129,B 9.2202,C 0.1061,E1 9.1596,E2 338.0448} C_DIS
LIN {X -57.5634,Y 128.8705,Z 170,A 115.0741,B 9.2202,C 0.108,E1 9.1556,E2 336.4854} C_DIS
LIN {X -60.7185,Y 127.4144,Z 170,A 116.5232,B 9.2202,C 0.1091,E1 9.1519,E2 335.0325} C_DIS
LIN {X -63.8721,Y 125.8632,Z 170,A 117.9357,B 9.2201,C 0.1112,E1 9.1484,E2 333.623} C_DIS
LIN {X -67.2979,Y 124.0678,Z 170,A 119.6171,B 9.2201,C 0.1113,E1 9.1442,E2 331.9289} C_DIS
LIN {X -71.075,Y 121.9436,Z 170,A 121.3931,B 9.2201,C 0.1136,E1 9.1399,E2 330.1523} C_DIS
LIN {X -74.7779,Y 119.7081,Z 170,A 123.1594,B 9.2201,C 0.1161,E1 9.1357,E2 328.3861} C_DIS
LIN {X -78.4159,Y 117.357,Z 170,A 124.9137,B 9.2201,C 0.1191,E1 9.1316,E2 326.634} C_DIS
LIN {X -82.0165,Y 114.8696,Z 170,A 126.7155,B 9.22,C 0.1216,E1 9.1275,E2 324.8306} C_DIS
LIN {X -85.4997,Y 112.3014,Z 170,A 128.5089,B 9.22,C 0.124,E1 9.1235,E2 323.0341} C_DIS
LIN {X -88.8885,Y 109.6389,Z 170,A 130.2997,B 9.22,C 0.1265,E1 9.1196,E2 321.2397} C_DIS
LIN {X -92.2135,Y 106.8569,Z 170,A 132.0334,B 9.2199,C 0.1303,E1 9.1159,E2 319.511} C_DIS
LIN {X -95.4452,Y 103.9804,Z 170,A 133.8185,B 9.2199,C 0.1333,E1 9.1122,E2 317.724} C_DIS
LIN {X -98.5806,Y 101.0134,Z 170,A 135.6063,B 9.2198,C 0.1362,E1 9.1086,E2 315.9333} C_DIS
LIN {X -101.6975,Y 97.875,Z 170,A 137.4474,B 9.2198,C 0.1391,E1 9.105,E2 314.0882} C_DIS
LIN {X -104.6431,Y 94.7183,Z 170,A 139.1947,B 9.2197,C 0.143,E1 9.1017,E2 312.3433} C_DIS
LIN {X -107.7252,Y 91.198,Z 170,A 141.1044,B 9.2197,C 0.1471,E1 9.0982,E2 310.4342} C_DIS
LIN {X -110.4644,Y 87.8597,Z 170,A 142.8698,B 9.2195,C 0.1509,E1 9.0951,E2 308.669} C_DIS
LIN {X -113.1262,Y 84.4049,Z 170,A 144.6694,B 9.2195,C 0.1545,E1 9.0921,E2 306.8675} C_DIS
LIN {X -115.631,Y 80.9403,Z 170,A 146.453,B 9.2195,C 0.1578,E1 9.0892,E2 305.0795} C_DIS
LIN {X -118.0889,Y 77.3101,Z 170,A 148.2442,B 9.2194,C 0.1619,E1 9.0864,E2 303.2887} C_DIS
LIN {X -120.3801,Y 73.6909,Z 170,A 149.9952,B 9.2193,C 0.166,E1 9.0838,E2 301.5379} C_DIS
LIN {X -122.6083,Y 69.9208,Z 170,A 151.7888,B 9.2193,C 0.1703,E1 9.0813,E2 299.7442} C_DIS
LIN {X -124.6937,Y 66.1283,Z 170,A 153.4838,B 9.2191,C 0.1759,E1 9.0791,E2 298.0589} C_DIS
LIN {X -126.4576,Y 62.6873,Z 170,A 155.0975,B 9.2191,C 0.1792,E1 9.077,E2 296.4412} C_DIS
LIN {X -127.9567,Y 59.5681,Z 170,A 156.5232,B 9.219,C 0.1826,E1 9.0753,E2 295.0143} C_DIS
LIN {X -129.4024,Y 56.3588,Z 170,A 157.9453,B 9.2189,C 0.1865,E1 9.0737,E2 293.5946} C_DIS
LIN {X -130.7493,Y 53.1598,Z 170,A 159.4055,B 9.2189,C 0.1894,E1 9.0722,E2 292.1293} C_DIS
LIN {X -131.977,Y 50.0356,Z 170,A 160.7897,B 9.2188,C 0.1928,E1 9.0708,E2 290.7438} C_DIS
LIN {X -133.165,Y 46.7825,Z 170,A 162.2492,B 9.2188,C 0.1957,E1 9.0694,E2 289.2789} C_DIS
LIN {X -134.2728,Y 43.501,Z 170,A 163.6778,B 9.2186,C 0.1992,E1 9.0681,E2 287.8489} C_DIS
LIN {X -135.3293,Y 40.0921,Z 170,A 165.1199,B 9.2186,C 0.2033,E1 9.067,E2 286.4091} C_DIS
LIN {X -136.4807,Y 35.9778,Z 170,A 166.8782,B 9.2184,C 0.2078,E1 9.0657,E2 284.6495} C_DIS
LIN {X -137.3244,Y 32.6107,Z 170,A 168.4354,B 9.2184,C 0.2092,E1 9.0646,E2 283.0747} C_DIS
LIN {X -138.2549,Y 28.4059,Z 170,A 170.0918,B 9.2183,C 0.2158,E1 9.0637,E2 281.4319} C_DIS
LIN {X -138.9302,Y 24.8924,Z 170,A 171.5441,B 9.2182,C 0.22,E1 9.0629,E2 279.981} C_DIS
LIN {X -139.4825,Y 21.5841,Z 170,A 172.9446,B 9.2181,C 0.2232,E1 9.0623,E2 278.5769} C_DIS
LIN {X -139.9669,Y 18.1813,Z 170,A 174.3743,B 9.2181,C 0.2266,E1 9.0618,E2 277.1441} C_DIS
LIN {X -140.3824,Y 14.6377,Z 170,A 175.8507,B 9.2179,C 0.2303,E1 9.0613,E2 275.6656} C_DIS
LIN {X -140.7146,Y 11.0104,Z 170,A 177.3261,B 9.2179,C 0.2347,E1 9.061,E2 274.1921} C_DIS
LIN {X -140.9321,Y 7.7368,Z 170,A 178.712,B 9.2177,C 0.2376,E1 9.0608,E2 272.8006} C_DIS
LIN {X -141.1011,Y 3.4624,Z 170,A -179.5579,B 9.2176,C 0.2428,E1 9.0606,E2 271.0729} C_DIS
LIN {X -141.1448,Y -0.2138,Z 170,A -178.0314,B 9.2175,C 0.2465,E1 9.0606,E2 269.5434} C_DIS
LIN {X -141.0783,Y -4.2854,Z 170,A -176.3207,B 9.2174,C 0.2503,E1 9.0606,E2 267.8269} C_DIS
LIN {X -140.9197,Y -7.9655,Z 170,A -174.8425,B 9.2173,C 0.2549,E1 9.0609,E2 266.3523} C_DIS
LIN {X -140.6628,Y -11.6323,Z 170,A -173.4253,B 9.2171,C 0.2606,E1 9.0612,E2 264.946} C_DIS
LIN {X -140.3824,Y -14.6384,Z 170,A -171.9765,B 9.2171,C 0.2602,E1 9.0616,E2 263.4695} C_DIS
LIN {X -139.9659,Y -18.1887,Z 170,A -170.5852,B 9.217,C 0.2654,E1 9.0621,E2 262.0872} C_DIS
LIN {X -139.4774,Y -21.6175,Z 170,A -169.1596,B 9.2169,C 0.269,E1 9.0627,E2 260.6602} C_DIS
LIN {X -138.9231,Y -24.9321,Z 170,A -167.7586,B 9.2168,C 0.2723,E1 9.0633,E2 259.2556} C_DIS
LIN {X -138.2486,Y -28.4366,Z 170,A -166.3043,B 9.2167,C 0.2763,E1 9.0641,E2 257.8019} C_DIS
LIN {X -137.5095,Y -31.8203,Z 170,A -164.8761,B 9.2166,C 0.2799,E1 9.065,E2 256.3719} C_DIS
LIN {X -136.6844,Y -35.1971,Z 170,A -163.4517,B 9.2164,C 0.2836,E1 9.066,E2 254.9469} C_DIS
LIN {X -135.8108,Y -38.4294,Z 170,A -162.029,B 9.2164,C 0.2862,E1 9.067,E2 253.517} C_DIS
LIN {X -134.552,Y -42.627,Z 170,A -160.2524,B 9.2162,C 0.2911,E1 9.0685,E2 251.7421} C_DIS
LIN {X -133.4505,Y -45.9591,Z 170,A -158.8161,B 9.2161,C 0.2948,E1 9.0698,E2 250.3054} C_DIS
LIN {X -132.2978,Y -49.1792,Z 170,A -157.3985,B 9.216,C 0.298,E1 9.0711,E2 248.885} C_DIS
LIN {X -131.0539,Y -52.4043,Z 170,A -155.8805,B 9.216,C 0.2997,E1 9.0727,E2 247.353} C_DIS
LIN {X -129.3035,Y -56.5875,Z 170,A -153.9715,B 9.2158,C 0.3033,E1 9.0748,E2 245.4364} C_DIS
LIN {X -127.5913,Y -60.3483,Z 170,A -152.4077,B 9.2156,C 0.3097,E1 9.0766,E2 243.8886} C_DIS
LIN {X -126.073,Y -63.4599,Z 170,A -150.8744,B 9.2156,C 0.311,E1 9.0786,E2 242.3395} C_DIS
LIN {X -124.067,Y -67.2993,Z 170,A -149.1101,B 9.2154,C 0.3154,E1 9.0809,E2 240.5756} C_DIS
LIN {X -121.9461,Y -71.0706,Z 170,A -147.3259,B 9.2153,C 0.3192,E1 9.0834,E2 238.7888} C_DIS
LIN {X -119.659,Y -74.8569,Z 170,A -145.5215,B 9.2151,C 0.3234,E1 9.086,E2 236.9842} C_DIS
LIN {X -117.356,Y -78.4174,Z 170,A -143.7867,B 9.2151,C 0.3272,E1 9.0887,E2 235.2486} C_DIS
LIN {X -114.8966,Y -81.9787,Z 170,A -141.9954,B 9.2149,C 0.3307,E1 9.0915,E2 233.4537} C_DIS
LIN {X -112.3292,Y -85.4633,Z 170,A -140.1949,B 9.2148,C 0.3338,E1 9.0946,E2 231.6483} C_DIS
LIN {X -109.6534,Y -88.8704,Z 170,A -138.3813,B 9.2147,C 0.3367,E1 9.0977,E2 229.8283} C_DIS
LIN {X -106.6047,Y -92.5057,Z 170,A -136.463,B 9.2145,C 0.3409,E1 9.1012,E2 227.9118} C_DIS
LIN {X -103.7192,Y -95.7293,Z 170,A -134.6987,B 9.2144,C 0.3444,E1 9.1045,E2 226.1471} C_DIS
LIN {X -100.4168,Y -99.1884,Z 170,A -132.7227,B 9.2143,C 0.3477,E1 9.1084,E2 224.1672} C_DIS
LIN {X -97.3251,Y -102.2234,Z 170,A -130.9588,B 9.2141,C 0.351,E1 9.1119,E2 222.4033} C_DIS
LIN {X -93.9179,Y -105.3624,Z 170,A -129.1168,B 9.214,C 0.3553,E1 9.1157,E2 220.5669} C_DIS
LIN {X -90.8713,Y -108.0007,Z 170,A -127.4047,B 9.214,C 0.3567,E1 9.1194,E2 218.8451} C_DIS
LIN {X -87.5174,Y -110.7366,Z 170,A -125.6213,B 9.2138,C 0.3593,E1 9.1233,E2 217.0588} C_DIS
LIN {X -84.0548,Y -113.3869,Z 170,A -123.8445,B 9.2138,C 0.3621,E1 9.1272,E2 215.2814} C_DIS
LIN {X -80.5483,Y -115.9038,Z 170,A -122.0957,B 9.2136,C 0.3649,E1 9.1312,E2 213.5333} C_DIS
LIN {X -76.9674,Y -118.3121,Z 170,A -120.3225,B 9.2136,C 0.3671,E1 9.1354,E2 211.7574} C_DIS
LIN {X -73.3043,Y -120.6163,Z 170,A -118.5322,B 9.2134,C 0.369,E1 9.1396,E2 209.9629} C_DIS
LIN {X -69.5577,Y -122.8154,Z 170,A -116.7582,B 9.2134,C 0.3712,E1 9.1439,E2 208.1877} C_DIS
LIN {X -66.1158,Y -124.7003,Z 170,A -115.267,B 9.2132,C 0.3752,E1 9.1476,E2 206.71} C_DIS
LIN {X -62.6752,Y -126.4636,Z 170,A -113.6665,B 9.2132,C 0.3765,E1 9.1516,E2 205.1053} C_DIS
LIN {X -59.5643,Y -127.9585,Z 170,A -112.2535,B 9.2131,C 0.3778,E1 9.1551,E2 203.6907} C_DIS
LIN {X -56.3548,Y -129.4041,Z 170,A -110.8472,B 9.2131,C 0.3798,E1 9.1587,E2 202.2874} C_DIS
LIN {X -53.1619,Y -130.7484,Z 170,A -109.4026,B 9.213,C 0.3804,E1 9.1625,E2 200.8376} C_DIS
LIN {X -50.0369,Y -131.9765,Z 170,A -108.0318,B 9.213,C 0.3816,E1 9.166,E2 199.4657} C_DIS
LIN {X -46.7834,Y -133.1647,Z 170,A -106.5878,B 9.213,C 0.382,E1 9.1698,E2 198.0165} C_DIS
LIN {X -43.5017,Y -134.2726,Z 170,A -105.1402,B 9.213,C 0.3823,E1 9.1737,E2 196.5632} C_DIS
LIN {X -39.9331,Y -135.3759,Z 170,A -103.5692,B 9.213,C 0.3823,E1 9.1779,E2 194.9846} C_DIS
LIN {X -35.958,Y -136.4859,Z 170,A -102.0046,B 9.2128,C 0.3856,E1 9.1821,E2 193.4344} C_DIS
LIN {X -32.6034,Y -137.3261,Z 170,A -100.5982,B 9.2128,C 0.3864,E1 9.1859,E2 192.0273} C_DIS
LIN {X -28.9036,Y -138.1536,Z 170,A -98.9202,B 9.2128,C 0.3842,E1 9.1905,E2 190.3305} C_DIS
LIN {X -24.9285,Y -138.9238,Z 170,A -97.4224,B 9.2127,C 0.3879,E1 9.1946,E2 188.8515} C_DIS
LIN {X -21.6177,Y -139.4773,Z 170,A -96.0377,B 9.2127,C 0.3879,E1 9.1984,E2 187.4634} C_DIS
LIN {X -18.187,Y -139.9661,Z 170,A -94.6202,B 9.2127,C 0.3881,E1 9.2024,E2 186.0441} C_DIS
LIN {X -14.6432,Y -140.3818,Z 170,A -93.1649,B 9.2127,C 0.3882,E1 9.2064,E2 184.5873} C_DIS
LIN {X -10.7972,Y -140.7302,Z 170,A -91.6955,B 9.2126,C 0.3905,E1 9.2105,E2 183.1303} C_DIS
LIN {X -7.7375,Y -140.9321,Z 170,A -90.3471,B 9.2126,C 0.3884,E1 9.2143,E2 181.7677} C_DIS
LIN {X -3.4605,Y -141.1012,Z 170,A -88.6454,B 9.2126,C 0.3891,E1 9.219,E2 180.0699} C_DIS
LIN {X 0.0005,Y -141.145,Z 170,A -87.2003,B 9.2126,C 0.3881,E1 9.2231,E2 178.619} C_DIS
LIN {X 0.0005,Y -141.145,Z 170,A -87.2003,B 9.2126,C 0.3881,E1 9.2231,E2 178.619} C_DIS
Enddeposition()
LIN {X 0.9578,Y -132.1891,Z 171,A -87.6181,B 9.2728,C 0.3483,E1 9.2812,E2 178.7807} C_DIS
Startdeposition()
$VEL.CP = VEL_PRINT
LIN {X -1.6404,Y -132.1862,Z 171,A -89.0033,B 9.2726,C 0.3535,E1 9.2772,E2 180.198} C_DIS
LIN {X -6.0328,Y -132.0588,Z 171,A -90.912,B 9.2726,C 0.3535,E1 9.2719,E2 182.108} C_DIS
LIN {X -10.1953,Y -131.8026,Z 171,A -92.7557,B 9.2726,C 0.3541,E1 9.2667,E2 183.9568} C_DIS
LIN {X -14.5678,Y -131.3906,Z 171,A -94.4924,B 9.2728,C 0.3506,E1 9.262,E2 185.674} C_DIS
LIN {X -17.7942,Y -130.9934,Z 171,A -95.9005,B 9.2728,C 0.3502,E1 9.2581,E2 187.0825} C_DIS
LIN {X -21.4675,Y -130.4405,Z 171,A -97.3703,B 9.2728,C 0.347,E1 9.254,E2 188.5358} C_DIS
LIN {X -24.6579,Y -129.875,Z 171,A -98.9358,B 9.2728,C 0.3495,E1 9.2497,E2 190.1213} C_DIS
LIN {X -27.8364,Y -129.2309,Z 171,A -100.3434,B 9.2728,C 0.3489,E1 9.2458,E2 191.5295} C_DIS
LIN {X -30.5521,Y -128.6166,Z 171,A -101.5568,B 9.2728,C 0.3484,E1 9.2425,E2 192.744} C_DIS
LIN {X -33.7444,Y -127.8158,Z 171,A -102.9836,B 9.2728,C 0.3475,E1 9.2387,E2 194.1711} C_DIS
LIN {X -36.8493,Y -126.9554,Z 171,A -104.3858,B 9.2729,C 0.3467,E1 9.2349,E2 195.5743} C_DIS
LIN {X -39.9396,Y -126.0173,Z 171,A -105.7911,B 9.2729,C 0.3458,E1 9.2312,E2 196.9805} C_DIS
LIN {X -43.6382,Y -124.7849,Z 171,A -107.4646,B 9.2729,C 0.3441,E1 9.2267,E2 198.6523} C_DIS
LIN {X -46.5038,Y -123.7451,Z 171,A -108.8178,B 9.273,C 0.3435,E1 9.2232,E2 200.0095} C_DIS
LIN {X -49.5216,Y -122.5686,Z 171,A -110.3142,B 9.273,C 0.3438,E1 9.2193,E2 201.5172} C_DIS
LIN {X -53.5735,Y -120.8532,Z 171,A -112.1444,B 9.2731,C 0.3404,E1 9.2146,E2 203.3383} C_DIS
LIN {X -56.871,Y -119.3361,Z 171,A -113.7846,B 9.2731,C 0.3399,E1 9.2104,E2 204.9865} C_DIS
LIN {X -59.9488,Y -117.82,Z 171,A -115.0663,B 9.2734,C 0.3344,E1 9.2073,E2 206.2434} C_DIS
LIN {X -62.7082,Y -116.3772,Z 171,A -116.5937,B 9.2733,C 0.3359,E1 9.2035,E2 207.7924} C_DIS
LIN {X -65.5725,Y -114.7876,Z 171,A -118.0165,B 9.2733,C 0.3341,E1 9.2,E2 209.2154} C_DIS
LIN {X -67.9639,Y -113.3885,Z 171,A -119.3083,B 9.2733,C 0.3341,E1 9.1969,E2 210.5181} C_DIS
LIN {X -70.7276,Y -111.6852,Z 171,A -120.7442,B 9.2734,C 0.3326,E1 9.1935,E2 211.9574} C_DIS
LIN {X -74.4307,Y -109.2528,Z 171,A -122.6836,B 9.2735,C 0.33,E1 9.189,E2 213.8988} C_DIS
LIN {X -77.7398,Y -106.9229,Z 171,A -124.3704,B 9.2736,C 0.326,E1 9.1851,E2 215.5772} C_DIS
LIN {X -80.6902,Y -104.7147,Z 171,A -126.0169,B 9.2737,C 0.3242,E1 9.1815,E2 217.2294} C_DIS
LIN {X -83.8687,Y -102.1863,Z 171,A -127.8595,B 9.2737,C 0.3226,E1 9.1774,E2 219.0814} C_DIS
LIN {X -87.1372,Y -99.4139,Z 171,A -129.7401,B 9.2739,C 0.3196,E1 9.1735,E2 220.9643} C_DIS
LIN {X -90.4011,Y -96.4559,Z 171,A -131.6527,B 9.2739,C 0.3161,E1 9.1695,E2 222.8767} C_DIS
LIN {X -93.4797,Y -93.4755,Z 171,A -133.5704,B 9.2741,C 0.3135,E1 9.1657,E2 224.8011} C_DIS
LIN {X -96.4686,Y -90.3875,Z 171,A -135.4334,B 9.2742,C 0.3097,E1 9.1621,E2 226.6634} C_DIS
LIN {X -99.4113,Y -87.1402,Z 171,A -137.3302,B 9.2743,C 0.3057,E1 9.1586,E2 228.5592} C_DIS
LIN {X -102.2032,Y -83.8481,Z 171,A -139.2364,B 9.2744,C 0.3022,E1 9.1552,E2 230.4688} C_DIS
LIN {X -104.8472,Y -80.5175,Z 171,A -141.1069,B 9.2746,C 0.2986,E1 9.152,E2 232.3418} C_DIS
LIN {X -107.4133,Y -77.0608,Z 171,A -142.8732,B 9.2748,C 0.2926,E1 9.1491,E2 234.0953} C_DIS
LIN {X -109.2669,Y -74.4098,Z 171,A -144.4433,B 9.2748,C 0.2922,E1 9.1465,E2 235.6847} C_DIS
LIN {X -111.6874,Y -70.7241,Z 171,A -146.3275,B 9.2749,C 0.2872,E1 9.1437,E2 237.5647} C_DIS
LIN {X -113.3916,Y -67.9587,Z 171,A -147.7292,B 9.275,C 0.2836,E1 9.1417,E2 238.9649} C_DIS
LIN {X -115.0352,Y -65.1385,Z 171,A -149.2051,B 9.2751,C 0.2812,E1 9.1396,E2 240.4473} C_DIS
LIN {X -116.8103,Y -61.8952,Z 171,A -150.5986,B 9.2753,C 0.2737,E1 9.1378,E2 241.8147} C_DIS
LIN {X -118.327,Y -58.944,Z 171,A -152.0651,B 9.2754,C 0.2705,E1 9.1359,E2 243.2838} C_DIS
LIN {X -119.4993,Y -56.5296,Z 171,A -153.4337,B 9.2754,C 0.2709,E1 9.1343,E2 244.6761} C_DIS
LIN {X -121.0458,Y -53.1403,Z 171,A -154.9938,B 9.2756,C 0.2658,E1 9.1325,E2 246.2286} C_DIS
LIN {X -122.5684,Y -49.5219,Z 171,A -156.8108,B 9.2756,C 0.2631,E1 9.1305,E2 248.0581} C_DIS
LIN {X -123.9141,Y -46.0525,Z 171,A -158.365,B 9.2758,C 0.2578,E1 9.129,E2 249.6042} C_DIS
LIN {X -125.0055,Y -43.0018,Z 171,A -159.8338,B 9.2758,C 0.2551,E1 9.1276,E2 251.0796} C_DIS
LIN {X -126.3968,Y -38.7209,Z 171,A -161.5327,B 9.2761,C 0.2456,E1 9.1262,E2 252.7471} C_DIS
LIN {X -127.1175,Y -36.292,Z 171,A -162.8824,B 9.2761,C 0.2467,E1 9.1251,E2 254.1259} C_DIS
LIN {X -127.9598,Y -33.2001,Z 171,A -164.2973,B 9.2761,C 0.2433,E1 9.1241,E2 255.5429} C_DIS
LIN {X -128.8808,Y -29.4145,Z 171,A -166.0763,B 9.2762,C 0.24,E1 9.123,E2 257.3311} C_DIS
LIN {X -129.6528,Y -25.8062,Z 171,A -167.7319,B 9.2763,C 0.2363,E1 9.122,E2 258.9922} C_DIS
LIN {X -130.2432,Y -22.6417,Z 171,A -169.186,B 9.2764,C 0.2333,E1 9.1213,E2 260.452} C_DIS
LIN {X -130.8318,Y -18.9369,Z 171,A -170.7109,B 9.2766,C 0.2271,E1 9.1207,E2 261.9635} C_DIS
LIN {X -131.3175,Y -15.2129,Z 171,A -172.4971,B 9.2766,C 0.2249,E1 9.1201,E2 263.7671} C_DIS
LIN {X -131.7079,Y -11.3408,Z 171,A -174.1595,B 9.2767,C 0.2197,E1 9.1196,E2 265.425} C_DIS
LIN {X -131.9749,Y -7.6421,Z 171,A -175.6918,B 9.2769,C 0.2138,E1 9.1194,E2 266.9471} C_DIS
LIN {X -132.1429,Y -3.7166,Z 171,A -177.2385,B 9.2771,C 0.2064,E1 9.1192,E2 268.4737} C_DIS
LIN {X -132.1988,Y 0.0839,Z 171,A -179.1789,B 9.2771,C 0.2063,E1 9.1192,E2 270.4473} C_DIS
LIN {X -132.143,Y 3.7116,Z 171,A 179.184,B 9.2771,C 0.2027,E1 9.1192,E2 272.0903} C_DIS
LIN {X -131.9464,Y 8.1045,Z 171,A 177.2872,B 9.2773,C 0.197,E1 9.1195,E2 273.9842} C_DIS
LIN {X -131.6177,Y 12.3451,Z 171,A 175.4362,B 9.2773,C 0.1918,E1 9.1199,E2 275.8344} C_DIS
LIN {X -131.2018,Y 16.1826,Z 171,A 173.7878,B 9.2775,C 0.1866,E1 9.1205,E2 277.4782} C_DIS
LIN {X -130.6855,Y 19.9223,Z 171,A 172.0908,B 9.2775,C 0.1828,E1 9.1211,E2 279.1808} C_DIS
LIN {X -130.2356,Y 22.6841,Z 171,A 170.7604,B 9.2775,C 0.1812,E1 9.1218,E2 280.5237} C_DIS
LIN {X -129.5594,Y 26.2651,Z 171,A 169.279,B 9.2777,C 0.1751,E1 9.1226,E2 281.992} C_DIS
LIN {X -128.8753,Y 29.4388,Z 171,A 167.7546,B 9.2777,C 0.173,E1 9.1235,E2 283.5288} C_DIS
LIN {X -127.8277,Y 33.7,Z 171,A 165.9109,B 9.2778,C 0.1667,E1 9.1247,E2 285.3636} C_DIS
LIN {X -126.9633,Y 36.8224,Z 171,A 164.4852,B 9.2779,C 0.1631,E1 9.1258,E2 286.7904} C_DIS
LIN {X -126.0226,Y 39.9231,Z 171,A 163.0596,B 9.2779,C 0.1595,E1 9.127,E2 288.2171} C_DIS
LIN {X -124.8539,Y 43.4393,Z 171,A 161.4283,B 9.278,C 0.1554,E1 9.1285,E2 289.8497} C_DIS
LIN {X -123.7522,Y 46.4847,Z 171,A 159.9997,B 9.278,C 0.152,E1 9.1299,E2 291.2797} C_DIS
LIN {X -122.5688,Y 49.521,Z 171,A 158.4811,B 9.2781,C 0.1498,E1 9.1314,E2 292.8093} C_DIS
LIN {X -120.8494,Y 53.5819,Z 171,A 156.633,B 9.2782,C 0.1437,E1 9.1335,E2 294.6481} C_DIS
LIN {X -119.299,Y 56.9489,Z 171,A 154.9983,B 9.2782,C 0.1399,E1 9.1354,E2 296.2843} C_DIS
LIN {X -117.8668,Y 59.8568,Z 171,A 153.7333,B 9.2784,C 0.1339,E1 9.137,E2 297.5315} C_DIS
LIN {X -116.5517,Y 62.3833,Z 171,A 152.2285,B 9.2784,C 0.1351,E1 9.139,E2 299.0666} C_DIS
LIN {X -114.7663,Y 65.6098,Z 171,A 150.6994,B 9.2784,C 0.1299,E1 9.141,E2 300.586} C_DIS
LIN {X -113.3771,Y 67.983,Z 171,A 149.4858,B 9.2784,C 0.1273,E1 9.1428,E2 301.801} C_DIS
LIN {X -111.6837,Y 70.7299,Z 171,A 147.984,B 9.2784,C 0.1255,E1 9.145,E2 303.3133} C_DIS
LIN {X -109.2835,Y 74.3852,Z 171,A 146.0495,B 9.2785,C 0.1215,E1 9.148,E2 305.2505} C_DIS
LIN {X -107.1616,Y 77.4105,Z 171,A 144.4279,B 9.2785,C 0.118,E1 9.1506,E2 306.8727} C_DIS
LIN {X -104.7173,Y 80.6868,Z 171,A 142.619,B 9.2786,C 0.1144,E1 9.1537,E2 308.6841} C_DIS
LIN {X -102.0343,Y 84.0538,Z 171,A 140.721,B 9.2786,C 0.1107,E1 9.157,E2 310.584} C_DIS
LIN {X -99.4141,Y 87.137,Z 171,A 138.946,B 9.2787,C 0.1071,E1 9.1603,E2 312.3597} C_DIS
LIN {X -96.4669,Y 90.3894,Z 171,A 137.0314,B 9.2787,C 0.1032,E1 9.1639,E2 314.2738} C_DIS
LIN {X -93.4693,Y 93.4858,Z 171,A 135.1228,B 9.2787,C 0.1,E1 9.1676,E2 316.1854} C_DIS
LIN {X -90.3947,Y 96.462,Z 171,A 133.2471,B 9.2788,C 0.0966,E1 9.1714,E2 318.0617} C_DIS
LIN {X -87.1429,Y 99.409,Z 171,A 131.3496,B 9.2788,C 0.0928,E1 9.1754,E2 319.9568} C_DIS
LIN {X -83.8581,Y 102.195,Z 171,A 129.4638,B 9.2788,C 0.0895,E1 9.1794,E2 321.843} C_DIS
LIN {X -80.5386,Y 104.8311,Z 171,A 127.5712,B 9.2789,C 0.0871,E1 9.1836,E2 323.7403} C_DIS
LIN {X -76.7828,Y 107.6121,Z 171,A 125.7313,B 9.2789,C 0.0805,E1 9.1877,E2 325.5568} C_DIS
LIN {X -73.7658,Y 109.7028,Z 171,A 123.9622,B 9.2789,C 0.0809,E1 9.1918,E2 327.3452} C_DIS
LIN {X -70.31,Y 111.9488,Z 171,A 122.2515,B 9.279,C 0.0767,E1 9.1958,E2 329.0455} C_DIS
LIN {X -67.953,Y 113.395,Z 171,A 121.0522,B 9.279,C 0.0749,E1 9.1987,E2 330.2438} C_DIS
LIN {X -65.156,Y 115.0252,Z 171,A 119.526,B 9.279,C 0.0749,E1 9.2024,E2 331.7831} C_DIS
LIN {X -61.9074,Y 116.8038,Z 171,A 118.132,B 9.279,C 0.069,E1 9.2058,E2 333.1512} C_DIS
LIN {X -59.4443,Y 118.0768,Z 171,A 116.7959,B 9.279,C 0.0697,E1 9.2091,E2 334.5019} C_DIS
LIN {X -56.5173,Y 119.5051,Z 171,A 115.3119,B 9.279,C 0.0692,E1 9.2129,E2 335.9932} C_DIS
LIN {X -53.085,Y 121.0696,Z 171,A 113.7439,B 9.279,C 0.066,E1 9.2169,E2 337.5522} C_DIS
LIN {X -49.4921,Y 122.5804,Z 171,A 111.9581,B 9.279,C 0.0658,E1 9.2215,E2 339.3478} C_DIS
LIN {X -46.048,Y 123.9158,Z 171,A 110.4241,B 9.2791,C 0.0629,E1 9.2255,E2 340.8727} C_DIS
LIN {X -43.001,Y 125.0058,Z 171,A 108.9712,B 9.2791,C 0.0624,E1 9.2293,E2 342.3304} C_DIS
LIN {X -38.8301,Y 126.3633,Z 171,A 107.3612,B 9.2791,C 0.0555,E1 9.2335,E2 343.9053} C_DIS
LIN {X -36.3933,Y 127.0889,Z 171,A 105.9867,B 9.2791,C 0.0595,E1 9.2373,E2 345.3108} C_DIS
LIN {X -33.2371,Y 127.9504,Z 171,A 104.5657,B 9.2791,C 0.0584,E1 9.2411,E2 346.7312} C_DIS
LIN {X -29.4033,Y 128.8834,Z 171,A 102.7925,B 9.2791,C 0.0584,E1 9.2459,E2 348.5105} C_DIS
LIN {X -25.7787,Y 129.6584,Z 171,A 101.1385,B 9.2791,C 0.0583,E1 9.2505,E2 350.1691} C_DIS
LIN {X -22.5943,Y 130.2517,Z 171,A 99.6886,B 9.2791,C 0.0583,E1 9.2545,E2 351.6235} C_DIS
LIN {X -18.9328,Y 130.8324,Z 171,A 98.2203,B 9.2791,C 0.0551,E1 9.2585,E2 353.0746} C_DIS
LIN {X -15.5723,Y 131.2746,Z 171,A 96.7785,B 9.2791,C 0.054,E1 9.2625,E2 354.5124} C_DIS
LIN {X -12.4765,Y 131.6051,Z 171,A 95.2915,B 9.2791,C 0.0561,E1 9.2666,E2 356.0147} C_DIS
LIN {X -8.1011,Y 131.9467,Z 171,A 93.4404,B 9.2791,C 0.0547,E1 9.2718,E2 357.8589} C_DIS
LIN {X -3.7111,Y 132.1431,Z 171,A 91.5274,B 9.2791,C 0.0547,E1 9.2771,E2 359.7719} C_DIS
LIN {X 0.4844,Y 132.1945,Z 171,A 89.9035,B 9.2791,C 0.0509,E1 9.2816,E2 361.3723} C_DIS
LIN {X 3.7219,Y 132.1428,Z 171,A 88.4696,B 9.2791,C 0.0515,E1 9.2856,E2 362.8092} C_DIS
LIN {X 6.4913,Y 132.0357,Z 171,A 87.1283,B 9.2791,C 0.0543,E1 9.2894,E2 364.1663} C_DIS
LIN {X 10.1922,Y 131.8028,Z 171,A 85.402,B 9.2791,C 0.0568,E1 9.2942,E2 365.9059} C_DIS
LIN {X 14.574,Y 131.3899,Z 171,A 83.6656,B 9.2791,C 0.0541,E1 9.299,E2 367.6216} C_DIS
LIN {X 17.7986,Y 130.9928,Z 171,A 82.2631,B 9.2791,C 0.0544,E1 9.3029,E2 369.0231} C_DIS
LIN {X 21.4635,Y 130.4412,Z 171,A 80.8032,B 9.2791,C 0.0523,E1 9.3069,E2 370.4654} C_DIS
LIN {X 24.6571,Y 129.8751,Z 171,A 79.2434,B 9.2791,C 0.056,E1 9.3112,E2 372.0427} C_DIS
LIN {X 27.8428,Y 129.2295,Z 171,A 77.7966,B 9.2791,C 0.0575,E1 9.3152,E2 373.4936} C_DIS
LIN {X 31.7456,Y 128.3289,Z 171,A 75.9818,B 9.2791,C 0.0602,E1 9.3201,E2 375.3173} C_DIS
LIN {X 35.2823,Y 127.3999,Z 171,A 74.5327,B 9.2791,C 0.0587,E1 9.324,E2 376.7502} C_DIS
LIN {X 38.3851,Y 126.4996,Z 171,A 73.0017,B 9.2791,C 0.0624,E1 9.3281,E2 378.2962} C_DIS
LIN {X 41.9085,Y 125.376,Z 171,A 71.5413,B 9.2791,C 0.0609,E1 9.332,E2 379.7398} C_DIS
LIN {X 44.9797,Y 124.3072,Z 171,A 70.141,B 9.2791,C 0.0621,E1 9.3356,E2 381.1388} C_DIS
LIN {X 48.1562,Y 123.1117,Z 171,A 68.6981,B 9.2791,C 0.063,E1 9.3394,E2 382.5783} C_DIS
LIN {X 51.6584,Y 121.6858,Z 171,A 66.9222,B 9.2791,C 0.0676,E1 9.344,E2 384.3702} C_DIS
LIN {X 55.0497,Y 120.1881,Z 171,A 65.3417,B 9.2791,C 0.0689,E1 9.348,E2 385.9474} C_DIS
LIN {X 58.3979,Y 118.5964,Z 171,A 63.8579,B 9.2791,C 0.0684,E1 9.3517,E2 387.4168} C_DIS
LIN {X 60.8913,Y 117.3374,Z 171,A 62.68,B 9.2791,C 0.0693,E1 9.3546,E2 388.5909} C_DIS
LIN {X 64.157,Y 115.5848,Z 171,A 61.0597,B 9.2791,C 0.0718,E1 9.3586,E2 390.2131} C_DIS
LIN {X 66.9754,Y 113.9747,Z 171,A 59.773,B 9.2791,C 0.0713,E1 9.3617,E2 391.4857} C_DIS
LIN {X 69.6229,Y 112.3773,Z 171,A 58.385,B 9.2791,C 0.0743,E1 9.365,E2 392.8795} C_DIS
LIN {X 72.5271,Y 110.5251,Z 171,A 56.7368,B 9.279,C 0.0798,E1 9.3689,E2 394.5461} C_DIS
LIN {X 76.1307,Y 108.0744,Z 171,A 54.8802,B 9.279,C 0.0822,E1 9.3732,E2 396.3992} C_DIS
LIN {X 79.6213,Y 105.5291,Z 171,A 53.0393,B 9.279,C 0.0848,E1 9.3773,E2 398.2367} C_DIS
LIN {X 82.7901,Y 103.0621,Z 171,A 51.2932,B 9.279,C 0.088,E1 9.3811,E2 399.984} C_DIS
LIN {X 86.2221,Y 100.2082,Z 171,A 49.4512,B 9.2789,C 0.0896,E1 9.385,E2 401.8155} C_DIS
LIN {X 89.2098,Y 97.5585,Z 171,A 47.6768,B 9.2789,C 0.0938,E1 9.3887,E2 403.5956} C_DIS
LIN {X 92.3246,Y 94.6161,Z 171,A 45.8743,B 9.2789,C 0.0964,E1 9.3924,E2 405.3922} C_DIS
LIN {X 95.1997,Y 91.7227,Z 171,A 44.1584,B 9.2789,C 0.0989,E1 9.3957,E2 407.1026} C_DIS
LIN {X 97.9525,Y 88.7764,Z 171,A 42.3608,B 9.2788,C 0.1036,E1 9.3991,E2 408.9067} C_DIS
LIN {X 100.8149,Y 85.512,Z 171,A 40.501,B 9.2788,C 0.1072,E1 9.4025,E2 410.7647} C_DIS
LIN {X 103.5848,Y 82.1352,Z 171,A 38.6734,B 9.2787,C 0.1101,E1 9.4057,E2 412.5854} C_DIS
LIN {X 106.1807,Y 78.7506,Z 171,A 36.816,B 9.2787,C 0.1145,E1 9.4088,E2 414.4447} C_DIS
LIN {X 108.3542,Y 75.7324,Z 171,A 35.3238,B 9.2787,C 0.1157,E1 9.4112,E2 415.9236} C_DIS
LIN {X 110.5557,Y 72.4807,Z 171,A 33.5467,B 9.2785,C 0.1214,E1 9.414,E2 417.7104} C_DIS
LIN {X 112.794,Y 68.9456,Z 171,A 31.9265,B 9.2785,C 0.1216,E1 9.4164,E2 419.3088} C_DIS
LIN {X 114.2143,Y 66.5671,Z 171,A 30.6652,B 9.2785,C 0.1259,E1 9.4182,E2 420.578} C_DIS
LIN {X 116.0333,Y 63.3421,Z 171,A 28.9682,B 9.2784,C 0.132,E1 9.4205,E2 422.2869} C_DIS
LIN {X 118.083,Y 59.4322,Z 171,A 27.189,B 9.2784,C 0.1339,E1 9.4227,E2 424.0513} C_DIS
LIN {X 119.5051,Y 56.5174,Z 171,A 25.7418,B 9.2784,C 0.1385,E1 9.4245,E2 425.5044} C_DIS
LIN {X 121.0435,Y 53.1455,Z 171,A 24.2269,B 9.2783,C 0.1407,E1 9.4262,E2 427.0095} C_DIS
LIN {X 122.6017,Y 49.4395,Z 171,A 22.4453,B 9.2782,C 0.1462,E1 9.4281,E2 428.7968} C_DIS
LIN {X 123.9155,Y 46.0489,Z 171,A 20.9558,B 9.2782,C 0.1486,E1 9.4296,E2 430.2773} C_DIS
LIN {X 125.046,Y 42.8851,Z 171,A 19.4971,B 9.2781,C 0.1526,E1 9.4309,E2 431.7373} C_DIS
LIN {X 126.361,Y 38.8379,Z 171,A 17.9534,B 9.2781,C 0.151,E1 9.4322,E2 433.2465} C_DIS
LIN {X 127.0956,Y 36.3703,Z 171,A 16.6008,B 9.278,C 0.1594,E1 9.4333,E2 434.6283} C_DIS
LIN {X 127.9497,Y 33.2399,Z 171,A 15.2162,B 9.278,C 0.1628,E1 9.4343,E2 436.0114} C_DIS
LIN {X 128.8808,Y 29.4148,Z 171,A 13.4779,B 9.2778,C 0.1683,E1 9.4354,E2 437.7549} C_DIS
LIN {X 129.6564,Y 25.7886,Z 171,A 11.8581,B 9.2778,C 0.1731,E1 9.4363,E2 439.3775} C_DIS
LIN {X 130.2503,Y 22.6018,Z 171,A 10.4514,B 9.2776,C 0.1772,E1 9.437,E2 440.7857} C_DIS
LIN {X 130.8324,Y 18.9328,Z 171,A 8.952,B 9.2776,C 0.1793,E1 9.4377,E2 442.2732} C_DIS
LIN {X 131.2583,Y 15.7091,Z 171,A 7.6033,B 9.2776,C 0.182,E1 9.4381,E2 443.6159} C_DIS
LIN {X 131.6038,Y 12.4899,Z 171,A 6.1165,B 9.2774,C 0.188,E1 9.4385,E2 445.1139} C_DIS
LIN {X 131.9462,Y 8.1089,Z 171,A 4.2904,B 9.2774,C 0.1917,E1 9.4389,E2 446.9324} C_DIS
LIN {X 132.1433,Y 3.7024,Z 171,A 2.4078,B 9.2773,C 0.1966,E1 9.4391,E2 448.8132} C_DIS
LIN {X 132.1979,Y -0.2096,Z 171,A 0.777,B 9.2772,C 0.2001,E1 9.4391,E2 450.4379} C_DIS
LIN {X 132.1431,Y -3.7111,Z 171,A -0.7961,B 9.2771,C 0.2058,E1 9.4391,E2 452.019} C_DIS
LIN {X 131.9749,Y -7.6429,Z 171,A -2.486,B 9.277,C 0.2104,E1 9.4388,E2 453.7087} C_DIS
LIN {X 131.7073,Y -11.3484,Z 171,A -4.091,B 9.2769,C 0.2149,E1 9.4384,E2 455.3147} C_DIS
LIN {X 131.2571,Y -15.719,Z 171,A -5.9374,B 9.2768,C 0.2192,E1 9.4379,E2 457.156} C_DIS
LIN {X 130.7664,Y -19.3946,Z 171,A -7.5429,B 9.2767,C 0.2238,E1 9.4372,E2 458.7629} C_DIS
LIN {X 130.1635,Y -23.0871,Z 171,A -9.0116,B 9.2767,C 0.225,E1 9.4365,E2 460.2149} C_DIS
LIN {X 129.5619,Y -26.2527,Z 171,A -10.4113,B 9.2765,C 0.2291,E1 9.4358,E2 461.6164} C_DIS
LIN {X 128.8605,Y -29.5036,Z 171,A -11.886,B 9.2765,C 0.234,E1 9.4349,E2 463.0965} C_DIS
LIN {X 127.8222,Y -33.7204,Z 171,A -13.6605,B 9.2763,C 0.2369,E1 9.4337,E2 464.86} C_DIS
LIN {X 126.961,Y -36.8304,Z 171,A -15.0374,B 9.2763,C 0.2404,E1 9.4326,E2 466.2357} C_DIS
LIN {X 126.0232,Y -39.9213,Z 171,A -16.4152,B 9.2762,C 0.2438,E1 9.4315,E2 467.6123} C_DIS
LIN {X 124.8484,Y -43.455,Z 171,A -18.0067,B 9.276,C 0.2478,E1 9.4301,E2 469.2028} C_DIS
LIN {X 123.7458,Y -46.502,Z 171,A -19.3902,B 9.276,C 0.2512,E1 9.4287,E2 470.5852} C_DIS
LIN {X 122.5679,Y -49.5232,Z 171,A -20.8672,B 9.2758,C 0.2566,E1 9.4272,E2 472.0724} C_DIS
LIN {X 120.8414,Y -53.5998,Z 171,A -22.6592,B 9.2758,C 0.259,E1 9.4252,E2 473.851} C_DIS
LIN {X 119.2933,Y -56.9608,Z 171,A -24.3086,B 9.2756,C 0.2643,E1 9.4233,E2 475.5076} C_DIS
LIN {X 117.3416,Y -60.8834,Z 171,A -26.0912,B 9.2756,C 0.2667,E1 9.421,E2 477.2782} C_DIS
LIN {X 115.595,Y -64.1386,Z 171,A -27.6946,B 9.2754,C 0.271,E1 9.4189,E2 478.8836} C_DIS
LIN {X 113.9942,Y -66.9422,Z 171,A -28.9747,B 9.2754,C 0.2719,E1 9.4171,E2 480.1508} C_DIS
LIN {X 112.5472,Y -69.3479,Z 171,A -30.3863,B 9.2752,C 0.2793,E1 9.4151,E2 481.5873} C_DIS
LIN {X 110.4785,Y -72.5979,Z 171,A -32.0185,B 9.2751,C 0.2827,E1 9.4126,E2 483.2166} C_DIS
LIN {X 108.0771,Y -76.1268,Z 171,A -33.7434,B 9.2751,C 0.2844,E1 9.4099,E2 484.9284} C_DIS
LIN {X 105.9052,Y -79.1206,Z 171,A -35.3878,B 9.2749,C 0.2892,E1 9.4071,E2 486.5794} C_DIS
LIN {X 103.5687,Y -82.1554,Z 171,A -37.086,B 9.2747,C 0.294,E1 9.4042,E2 488.284} C_DIS
LIN {X 100.7501,Y -85.5883,Z 171,A -38.9441,B 9.2747,C 0.2969,E1 9.4009,E2 490.1359} C_DIS
LIN {X 97.9532,Y -88.7756,Z 171,A -40.781,B 9.2745,C 0.301,E1 9.3975,E2 491.9746} C_DIS
LIN {X 95.0175,Y -91.9109,Z 171,A -42.6177,B 9.2744,C 0.3045,E1 9.3939,E2 493.8101} C_DIS
LIN {X 91.8665,Y -95.0605,Z 171,A -44.5029,B 9.2743,C 0.3076,E1 9.3902,E2 495.6917} C_DIS
LIN {X 88.6079,Y -98.1054,Z 171,A -46.4632,B 9.2741,C 0.3122,E1 9.3862,E2 497.6573} C_DIS
LIN {X 85.5501,Y -100.7825,Z 171,A -48.1896,B 9.2741,C 0.3149,E1 9.3825,E2 499.3812} C_DIS
LIN {X 82.1369,Y -103.5834,Z 171,A -50.0128,B 9.274,C 0.3167,E1 9.3786,E2 501.1953} C_DIS
LIN {X 78.7485,Y -106.1823,Z 171,A -51.9001,B 9.2738,C 0.3208,E1 9.3743,E2 503.0887} C_DIS
LIN {X 75.7339,Y -108.3531,Z 171,A -53.3996,B 9.2738,C 0.3213,E1 9.371,E2 504.5763} C_DIS
LIN {X 72.4711,Y -110.562,Z 171,A -55.207,B 9.2736,C 0.3264,E1 9.3667,E2 506.3973} C_DIS
LIN {X 68.8815,Y -112.8334,Z 171,A -56.828,B 9.2736,C 0.3247,E1 9.363,E2 507.9933} C_DIS
LIN {X 66.5335,Y -114.2338,Z 171,A -58.088,B 9.2736,C 0.3282,E1 9.3599,E2 509.2635} C_DIS
LIN {X 63.3202,Y -116.0452,Z 171,A -59.7534,B 9.2734,C 0.332,E1 9.3558,E2 510.9383} C_DIS
LIN {X 60.885,Y -117.3407,Z 171,A -60.8758,B 9.2734,C 0.3322,E1 9.3531,E2 512.0529} C_DIS
LIN {X 57.9727,Y -118.8061,Z 171,A -62.2753,B 9.2734,C 0.3339,E1 9.3495,E2 513.4519} C_DIS
LIN {X 54.616,Y -120.3869,Z 171,A -63.8593,B 9.2734,C 0.3356,E1 9.3455,E2 515.0344} C_DIS
LIN {X 51.6506,Y -121.689,Z 171,A -65.4392,B 9.2731,C 0.341,E1 9.3414,E2 516.6368} C_DIS
LIN {X 47.5076,Y -123.3638,Z 171,A -67.1952,B 9.2731,C 0.3395,E1 9.3369,E2 518.3723} C_DIS
LIN {X 44.4414,Y -124.5013,Z 171,A -68.5898,B 9.2731,C 0.3406,E1 9.3333,E2 519.7653} C_DIS
LIN {X 40.9828,Y -125.6841,Z 171,A -70.343,B 9.2729,C 0.3458,E1 9.3286,E2 521.5402} C_DIS
LIN {X 37.9094,Y -126.645,Z 171,A -71.5592,B 9.273,C 0.3434,E1 9.3254,E2 522.7357} C_DIS
LIN {X 34.7979,Y -127.5349,Z 171,A -72.9568,B 9.273,C 0.3446,E1 9.3216,E2 524.1337} C_DIS
LIN {X 31.6595,Y -128.3497,Z 171,A -74.5234,B 9.2728,C 0.349,E1 9.3173,E2 525.7208} C_DIS
LIN {X 26.9878,Y -129.4124,Z 171,A -76.3546,B 9.2729,C 0.3456,E1 9.3124,E2 527.5235} C_DIS
LIN {X 23.719,Y -130.0504,Z 171,A -77.7141,B 9.2729,C 0.3449,E1 9.3087,E2 528.8738} C_DIS
LIN {X 20.5273,Y -130.5918,Z 171,A -79.2604,B 9.2729,C 0.3486,E1 9.3044,E2 530.4384} C_DIS
LIN {X 17.0381,Y -131.0925,Z 171,A -80.7262,B 9.2729,C 0.3481,E1 9.3003,E2 531.8975} C_DIS
LIN {X 14.1065,Y -131.4402,Z 171,A -82.0549,B 9.2728,C 0.3497,E1 9.2966,E2 533.2329} C_DIS
LIN {X 10.1868,Y -131.8032,Z 171,A -83.879,B 9.2727,C 0.3527,E1 9.2915,E2 535.0724} C_DIS
LIN {X 6.0086,Y -132.06,Z 171,A -85.7346,B 9.2727,C 0.354,E1 9.2863,E2 536.9339} C_DIS
LIN {X 1.6214,Y -132.1865,Z 171,A -87.5865,B 9.2727,C 0.3534,E1 9.2812,E2 538.7807} C_DIS
LIN {X 1.6214,Y -132.1865,Z 171,A -87.5865,B 9.2727,C 0.3534,E1 9.2812,E2 538.7807} C_DIS
Enddeposition()
LIN {X 0.9624,Y -133.1014,Z 171,A -87.5278,B 9.2725,C 0.3521,E1 9.2812,E2 538.7143} C_DIS
Startdeposition()
$VEL.CP = VEL_PRINT
LIN {X 3.1519,Y -133.0693,Z 171,A -86.0355,B 9.2729,C 0.341,E1 9.2855,E2 537.1537} C_DIS
LIN {X 7.4063,Y -132.9012,Z 171,A -84.2088,B 9.2729,C 0.3406,E1 9.2906,E2 535.3269} C_DIS
LIN {X 11.6069,Y -132.599,Z 171,A -82.5406,B 9.2728,C 0.3429,E1 9.2952,E2 533.6756} C_DIS
LIN {X 14.2448,Y -132.3409,Z 171,A -81.2825,B 9.2728,C 0.34,E1 9.2987,E2 532.4023} C_DIS
LIN {X 18.5709,Y -131.8037,Z 171,A -79.4859,B 9.2728,C 0.3407,E1 9.3036,E2 530.6145} C_DIS
LIN {X 22.0869,Y -131.2601,Z 171,A -77.9918,B 9.2728,C 0.3406,E1 9.3078,E2 529.1241} C_DIS
LIN {X 25.1639,Y -130.7051,Z 171,A -76.6073,B 9.2729,C 0.3389,E1 9.3116,E2 527.7339} C_DIS
LIN {X 29.3948,Y -129.8191,Z 171,A -74.7659,B 9.2729,C 0.3379,E1 9.3166,E2 525.8937} C_DIS
LIN {X 32.687,Y -129.0292,Z 171,A -73.3007,B 9.273,C 0.3366,E1 9.3206,E2 524.4265} C_DIS
LIN {X 36.4991,Y -128.0049,Z 171,A -71.6265,B 9.273,C 0.3356,E1 9.3251,E2 522.7543} C_DIS
LIN {X 39.8405,Y -127.0046,Z 171,A -69.9211,B 9.2733,C 0.3298,E1 9.3297,E2 521.0224} C_DIS
LIN {X 44.4093,Y -125.4806,Z 171,A -68.1073,B 9.2731,C 0.3331,E1 9.3344,E2 519.2393} C_DIS
LIN {X 49.336,Y -123.6249,Z 171,A -65.9776,B 9.2731,C 0.3334,E1 9.3399,E2 517.1247} C_DIS
LIN {X 53.0356,Y -122.0828,Z 171,A -64.1218,B 9.2733,C 0.3285,E1 9.3447,E2 515.2513} C_DIS
LIN {X 56.2285,Y -120.6459,Z 171,A -62.5981,B 9.2733,C 0.3261,E1 9.3486,E2 513.7243} C_DIS
LIN {X 61.4165,Y -118.0898,Z 171,A -60.2728,B 9.2733,C 0.3261,E1 9.3544,E2 511.4174} C_DIS
LIN {X 66.7835,Y -115.1409,Z 171,A -57.0248,B 9.274,C 0.3089,E1 9.3625,E2 508.091} C_DIS
LIN {X 70.5548,Y -112.8696,Z 171,A -55.6123,B 9.2737,C 0.3163,E1 9.3657,E2 506.7369} C_DIS
LIN {X 74.1273,Y -110.5562,Z 171,A -53.7495,B 9.2739,C 0.3125,E1 9.37,E2 504.8686} C_DIS
LIN {X 77.6614,Y -108.1029,Z 171,A -51.9281,B 9.2739,C 0.3099,E1 9.3742,E2 503.0493} C_DIS
LIN {X 81.1534,Y -105.5069,Z 171,A -49.7932,B 9.2742,C 0.3007,E1 9.379,E2 500.88} C_DIS
LIN {X 83.9725,Y -103.2772,Z 171,A -48.5033,B 9.2742,C 0.3034,E1 9.3817,E2 499.6207} C_DIS
LIN {X 87.3052,Y -100.4755,Z 171,A -46.6573,B 9.2742,C 0.3003,E1 9.3857,E2 497.7764} C_DIS
LIN {X 90.3553,Y -97.742,Z 171,A -44.3889,B 9.2747,C 0.2855,E1 9.3905,E2 495.4432} C_DIS
LIN {X 93.9949,Y -94.2469,Z 171,A -42.817,B 9.2745,C 0.2942,E1 9.3934,E2 493.944} C_DIS
LIN {X 96.9469,Y -91.2073,Z 171,A -40.9531,B 9.2746,C 0.2894,E1 9.397,E2 492.0732} C_DIS
LIN {X 99.3996,Y -88.5286,Z 171,A -38.784,B 9.2751,C 0.2723,E1 9.4012,E2 489.8271} C_DIS
LIN {X 103.0519,Y -84.2482,Z 171,A -37.2534,B 9.2747,C 0.2867,E1 9.4037,E2 488.405} C_DIS
LIN {X 105.0846,Y -81.6989,Z 171,A -35.6348,B 9.2749,C 0.2786,E1 9.4066,E2 486.7583} C_DIS
LIN {X 107.6413,Y -78.2997,Z 171,A -33.8666,B 9.275,C 0.2756,E1 9.4095,E2 484.9959} C_DIS
LIN {X 110.3796,Y -74.3899,Z 171,A -31.7956,B 9.2752,C 0.2702,E1 9.4128,E2 482.9208} C_DIS
LIN {X 112.8509,Y -70.5849,Z 171,A -29.8659,B 9.2753,C 0.2658,E1 9.4157,E2 480.9919} C_DIS
LIN {X 116.148,Y -65.0166,Z 171,A -27.1817,B 9.2754,C 0.261,E1 9.4194,E2 478.3174} C_DIS
LIN {X 118.0108,Y -61.567,Z 171,A -25.5915,B 9.2754,C 0.2588,E1 9.4215,E2 476.7374} C_DIS
LIN {X 119.5135,Y -58.5964,Z 171,A -24.1388,B 9.2756,C 0.2545,E1 9.4233,E2 475.2806} C_DIS
LIN {X 122.3225,Y -52.4813,Z 171,A -21.329,B 9.2758,C 0.2487,E1 9.4265,E2 472.4786} C_DIS
LIN {X 123.7603,Y -49.0001,Z 171,A -19.724,B 9.2758,C 0.2447,E1 9.4282,E2 470.874} C_DIS
LIN {X 124.9529,Y -45.8728,Z 171,A -18.1649,B 9.2761,C 0.238,E1 9.4297,E2 469.2988} C_DIS
LIN {X 126.8397,Y -40.3567,Z 171,A -15.8612,B 9.2761,C 0.2357,E1 9.4318,E2 467.0178} C_DIS
LIN {X 127.7533,Y -37.364,Z 171,A -13.953,B 9.2765,C 0.219,E1 9.4333,E2 465.0388} C_DIS
LIN {X 128.9715,Y -32.9145,Z 171,A -12.1005,B 9.2765,C 0.2165,E1 9.4346,E2 463.2008} C_DIS
LIN {X 129.9465,Y -28.8353,Z 171,A -10.6939,B 9.2765,C 0.2205,E1 9.4354,E2 461.8417} C_DIS
LIN {X 130.7566,Y -24.8941,Z 171,A -9.04,B 9.2765,C 0.2173,E1 9.4363,E2 460.1956} C_DIS
LIN {X 131.4893,Y -20.6804,Z 171,A -7.1618,B 9.2767,C 0.2111,E1 9.4372,E2 458.311} C_DIS
LIN {X 132.0807,Y -16.5004,Z 171,A -5.3081,B 9.2768,C 0.205,E1 9.4378,E2 456.451} C_DIS
LIN {X 132.522,Y -12.4512,Z 171,A -3.7138,B 9.2768,C 0.2036,E1 9.4383,E2 454.8744} C_DIS
LIN {X 132.8451,Y -8.322,Z 171,A -1.9803,B 9.277,C 0.1995,E1 9.4386,E2 453.1452} C_DIS
LIN {X 133.0262,Y -4.6261,Z 171,A -0.3532,B 9.277,C 0.1941,E1 9.4388,E2 451.5124} C_DIS
LIN {X 133.1071,Y -0.3858,Z 171,A 1.5226,B 9.2772,C 0.1876,E1 9.4388,E2 449.6288} C_DIS
LIN {X 133.0393,Y 4.2323,Z 171,A 3.3194,B 9.2772,C 0.1862,E1 9.4388,E2 447.8535} C_DIS
LIN {X 132.8589,Y 8.0973,Z 171,A 5.0553,B 9.2773,C 0.1798,E1 9.4385,E2 446.1074} C_DIS
LIN {X 132.4976,Y 12.7058,Z 171,A 6.979,B 9.2774,C 0.1755,E1 9.438,E2 444.19} C_DIS
LIN {X 132.1372,Y 16.0269,Z 171,A 8.3612,B 9.2774,C 0.1726,E1 9.4376,E2 442.8134} C_DIS
LIN {X 131.5753,Y 20.1252,Z 171,A 10.1246,B 9.2776,C 0.1679,E1 9.4369,E2 441.0505} C_DIS
LIN {X 130.9308,Y 23.967,Z 171,A 11.7465,B 9.2776,C 0.1644,E1 9.4361,E2 439.434} C_DIS
LIN {X 130.3651,Y 26.8711,Z 171,A 12.97,B 9.2776,C 0.1619,E1 9.4354,E2 438.2155} C_DIS
LIN {X 129.7624,Y 29.643,Z 171,A 14.2178,B 9.2777,C 0.1578,E1 9.4347,E2 436.9633} C_DIS
LIN {X 128.8377,Y 33.4416,Z 171,A 15.8505,B 9.2778,C 0.1543,E1 9.4336,E2 435.3356} C_DIS
LIN {X 127.9705,Y 36.6218,Z 171,A 17.6496,B 9.278,C 0.1417,E1 9.4322,E2 433.4889} C_DIS
LIN {X 126.9326,Y 40.0659,Z 171,A 18.6459,B 9.2779,C 0.1499,E1 9.4314,E2 432.5587} C_DIS
LIN {X 125.6454,Y 43.9353,Z 171,A 20.5979,B 9.278,C 0.1407,E1 9.4296,E2 430.5815} C_DIS
LIN {X 123.6069,Y 49.3804,Z 171,A 22.8236,B 9.278,C 0.1402,E1 9.4275,E2 428.3877} C_DIS
LIN {X 122.7651,Y 51.4361,Z 171,A 23.9356,B 9.2781,C 0.1341,E1 9.4262,E2 427.2561} C_DIS
LIN {X 121.3428,Y 54.7084,Z 171,A 25.4546,B 9.2781,C 0.1305,E1 9.4245,E2 425.7382} C_DIS
LIN {X 119.8643,Y 57.8772,Z 171,A 26.9133,B 9.2782,C 0.1276,E1 9.4228,E2 424.2841} C_DIS
LIN {X 118.2251,Y 61.1588,Z 171,A 28.6447,B 9.2783,C 0.1201,E1 9.4206,E2 422.5333} C_DIS
LIN {X 116.337,Y 64.6778,Z 171,A 30.2151,B 9.2783,C 0.1191,E1 9.4185,E2 420.9799} C_DIS
LIN {X 114.3526,Y 68.1245,Z 171,A 31.9431,B 9.2783,C 0.1145,E1 9.416,E2 419.2489} C_DIS
LIN {X 112.3791,Y 71.3338,Z 171,A 33.5667,B 9.2784,C 0.1105,E1 9.4136,E2 417.6242} C_DIS
LIN {X 109.9614,Y 75.0073,Z 171,A 35.4609,B 9.2784,C 0.106,E1 9.4107,E2 415.7289} C_DIS
LIN {X 107.2693,Y 78.8083,Z 171,A 37.2615,B 9.2784,C 0.1058,E1 9.4078,E2 413.9519} C_DIS
LIN {X 104.9601,Y 81.8595,Z 171,A 39.7478,B 9.2787,C 0.0836,E1 9.4033,E2 411.3631} C_DIS
LIN {X 101.2101,Y 86.4526,Z 171,A 41.5669,B 9.2787,C 0.0941,E1 9.4002,E2 409.6321} C_DIS
LIN {X 98.3015,Y 89.7464,Z 171,A 43.4778,B 9.2787,C 0.0896,E1 9.3966,E2 407.7181} C_DIS
LIN {X 94.1155,Y 94.1271,Z 171,A 45.9708,B 9.2787,C 0.0868,E1 9.3918,E2 405.238} C_DIS
LIN {X 91.2077,Y 96.9465,Z 171,A 47.7207,B 9.2787,C 0.0832,E1 9.3883,E2 403.4868} C_DIS
LIN {X 86.8519,Y 100.8672,Z 171,A 50.2269,B 9.2787,C 0.0787,E1 9.383,E2 400.9819} C_DIS
LIN {X 83.3121,Y 103.8106,Z 171,A 52.1978,B 9.2787,C 0.0754,E1 9.3788,E2 399.0119} C_DIS
LIN {X 79.2611,Y 106.9355,Z 171,A 54.1354,B 9.2787,C 0.0772,E1 9.3745,E2 397.1056} C_DIS
LIN {X 76.6767,Y 108.8032,Z 171,A 56.4757,B 9.2789,C 0.0544,E1 9.3689,E2 394.6483} C_DIS
LIN {X 71.611,Y 112.2023,Z 171,A 58.099,B 9.2789,C 0.0715,E1 9.3654,E2 393.1457} C_DIS
LIN {X 68.9013,Y 113.8862,Z 171,A 59.6697,B 9.2789,C 0.0653,E1 9.3616,E2 391.5513} C_DIS
LIN {X 65.0739,Y 116.1158,Z 171,A 61.5225,B 9.2789,C 0.0638,E1 9.3571,E2 389.7048} C_DIS
LIN {X 61.5863,Y 118.0006,Z 171,A 63.1968,B 9.2789,C 0.0621,E1 9.353,E2 388.0342} C_DIS
LIN {X 58.2105,Y 119.7039,Z 171,A 64.787,B 9.2789,C 0.0609,E1 9.349,E2 386.4486} C_DIS
LIN {X 55.6934,Y 120.8934,Z 171,A 66.0157,B 9.2789,C 0.0588,E1 9.3459,E2 385.2161} C_DIS
LIN {X 52.3875,Y 122.363,Z 171,A 67.5862,B 9.2789,C 0.0568,E1 9.3419,E2 383.6441} C_DIS
LIN {X 49.1244,Y 123.7102,Z 171,A 69.0315,B 9.2789,C 0.0567,E1 9.3382,E2 382.2079} C_DIS
LIN {X 45.8891,Y 124.947,Z 171,A 70.5167,B 9.2789,C 0.0553,E1 9.3343,E2 380.7235} C_DIS
Enddeposition()
END
